LIN {X 0,Y 197.202,Z 363.126,A -85,B 0,C 180,E1 -23005.854,E2 -23005.854} C_VEL
LIN {X 0,Y 193.789,Z 355.62,A -85,B 0,C 180,E1 -23008.882,E2 -23008.882} C_VEL
LIN {X 0,Y 191.136,Z 350.73,A -85,B 0,C 180,E1 -23011.177,E2 -23011.177} C_VEL
LIN {X 0,Y 188.874,Z 346.573,A -85,B 0,C 180,E1 -23013.258,E2 -23013.258} C_VEL
LIN {X 0,Y 185.862,Z 342.068,A -85,B 0,C 180,E1 -23016.015,E2 -23016.015} C_VEL
LIN {X 0,Y 185.125,Z 340.647,A -85,B 0,C 180,E1 -23016.804,E2 -23016.804} C_VEL
LIN {X 0,Y 182.731,Z 338.106,A -85,B 0,C 180,E1 -23019.16,E2 -23019.16} C_VEL
LIN {X 0,Y 181.419,Z 335.441,A -85,B 0,C 180,E1 -23020.775,E2 -23020.775} C_VEL
LIN {X 0,Y 178.641,Z 333.282,A -85,B 0,C 180,E1 -23024.014,E2 -23024.014} C_VEL
LIN {X 0,Y 177.261,Z 330.435,A -85,B 0,C 180,E1 -23026.384,E2 -23026.384} C_VEL
LIN {X 0,Y 177.054,Z 329.764,A -85,B 0,C 180,E1 -23026.806,E2 -23026.806} C_VEL
LIN {X 0,Y 172.985,Z 325.903,A -85,B 0,C 180,E1 -23040,E2 -23040} C_VEL
LIN {X 0,Y 177.156,Z 329.966,A -85,B 0,C 180,E1 -23053.259,E2 -23053.259} C_VEL
LIN {X 0,Y 178.201,Z 332.574,A -85,B 0,C 180,E1 -23055.146,E2 -23055.146} C_VEL
LIN {X 0,Y 181.712,Z 336.354,A -85,B 0,C 180,E1 -23059.486,E2 -23059.486} C_VEL
LIN {X 0,Y 183.271,Z 339.603,A -85,B 0,C 180,E1 -23061.364,E2 -23061.364} C_VEL
LIN {X 0,Y 185.721,Z 342.711,A -85,B 0,C 180,E1 -23063.781,E2 -23063.781} C_VEL
LIN {X 0,Y 187.904,Z 346.733,A -85,B 0,C 180,E1 -23065.921,E2 -23065.921} C_VEL
LIN {X 0,Y 189.084,Z 348.461,A -85,B 0,C 180,E1 -23066.957,E2 -23066.957} C_VEL
LIN {X 0,Y 191.285,Z 352.569,A -85,B 0,C 180,E1 -23068.957,E2 -23068.957} C_VEL
LIN {X 0,Y 194.891,Z 359.939,A -85,B 0,C 180,E1 -23072.134,E2 -23072.134} C_VEL
LIN {X 0,Y 198.257,Z 367.774,A -85,B 0,C 180,E1 -23075.122,E2 -23075.122} C_VEL
LIN {X 0,Y 200.917,Z 375.46,A -85,B 0,C 180,E1 -23077.724,E2 -23077.724} C_VEL
LIN {X 0,Y 202.539,Z 383.023,A -85,B 0,C 180,E1 -23079.938,E2 -23079.938} C_VEL
LIN {X 0,Y 203.603,Z 393.149,A -85,B 0,C 180,E1 -23082.673,E2 -23082.673} C_VEL
LIN {X 0,Y 203.75,Z 403.021,A -85,B 0,C 180,E1 -23085.29,E2 -23085.29} C_VEL
LIN {X 0,Y 203.187,Z 411.249,A -85,B 0,C 180,E1 -23087.478,E2 -23087.478} C_VEL
LIN {X 0,Y 198.333,Z 421.868,A -85,B 0,C 180,E1 -23089.707,E2 -23089.707} C_VEL
LIN {X 0,Y 193.072,Z 432.353,A -85,B 0,C 180,E1 -23092.431,E2 -23092.431} C_VEL
LIN {X 0,Y 187.527,Z 442.605,A -85,B 0,C 180,E1 -23095.794,E2 -23095.794} C_VEL
LIN {X 0,Y 183.46,Z 450.011,A -85,B 0,C 180,E1 -23098.858,E2 -23098.858} C_VEL
LIN {X 0,Y 179.707,Z 456.354,A -85,B 0,C 180,E1 -23102.011,E2 -23102.011} C_VEL
LIN {X 0,Y 175.598,Z 463.314,A -85,B 0,C 180,E1 -23106.407,E2 -23106.407} C_VEL
LIN {X 0,Y 172.589,Z 468.788,A -85,B 0,C 180,E1 -23110.987,E2 -23110.987} C_VEL
LIN {X 0,Y 170.443,Z 472.925,A -85,B 0,C 180,E1 -23115.675,E2 -23115.675} C_VEL
LIN {X 0,Y 169.294,Z 475.826,A -85,B 0,C 180,E1 -23120.441,E2 -23120.441} C_VEL
LIN {X 0,Y 168.85,Z 477.556,A -85,B 0,C 180,E1 -23125.224,E2 -23125.224} C_VEL
LIN {X 0,Y 168.868,Z 478.146,A -85,B 0,C 180,E1 -23129.999,E2 -23129.999} C_VEL
LIN {X 0,Y 168.811,Z 477.96,A -85,B 0,C 180,E1 -23132.539,E2 -23132.539} C_VEL
LIN {X 0,Y 168.123,Z 477.6,A -85,B 0,C 180,E1 -23134.528,E2 -23134.528} C_VEL
LIN {X 0,Y 165.469,Z 476.617,A -85,B 0,C 180,E1 -23137.794,E2 -23137.794} C_VEL
LIN {X 0,Y 163.446,Z 475.488,A -85,B 0,C 180,E1 -23140.46,E2 -23140.46} C_VEL
LIN {X 0,Y 162.86,Z 474.386,A -85,B 0,C 180,E1 -23142.503,E2 -23142.503} C_VEL
LIN {X 0,Y 162.958,Z 473.946,A -85,B 0,C 180,E1 -23143.184,E2 -23143.184} C_VEL
LIN {X 0,Y 165.212,Z 469.819,A -85,B 0,C 180,E1 -23148.604,E2 -23148.604} C_VEL
LIN {X 0,Y 168.096,Z 464.744,A -85,B 0,C 180,E1 -23153.315,E2 -23153.315} C_VEL
LIN {X 0,Y 172.217,Z 458.041,A -85,B 0,C 180,E1 -23157.988,E2 -23157.988} C_VEL
LIN {X 0,Y 176.662,Z 450.925,A -85,B 0,C 180,E1 -23161.809,E2 -23161.809} C_VEL
LIN {X 0,Y 181.724,Z 442.379,A -85,B 0,C 180,E1 -23165.457,E2 -23165.457} C_VEL
LIN {X 0,Y 187.448,Z 432.092,A -85,B 0,C 180,E1 -23168.902,E2 -23168.902} C_VEL
LIN {X 0,Y 192.941,Z 421.569,A -85,B 0,C 180,E1 -23171.662,E2 -23171.662} C_VEL
LIN {X 0,Y 197.1,Z 412.813,A -85,B 0,C 180,E1 -23173.545,E2 -23173.545} C_VEL
LIN {X 0,Y 197.872,Z 405.133,A -85,B 0,C 180,E1 -23175.704,E2 -23175.704} C_VEL
LIN {X 0,Y 197.933,Z 396.156,A -85,B 0,C 180,E1 -23178.212,E2 -23178.212} C_VEL
LIN {X 0,Y 197.384,Z 387.797,A -85,B 0,C 180,E1 -23180.576,E2 -23180.576} C_VEL
LIN {X 0,Y 196.151,Z 380.242,A -85,B 0,C 180,E1 -23182.871,E2 -23182.871} C_VEL
LIN {X 0,Y 193.642,Z 372.121,A -85,B 0,C 180,E1 -23185.768,E2 -23185.768} C_VEL
LIN {X 0,Y 190.07,Z 363.095,A -85,B 0,C 180,E1 -23189.442,E2 -23189.442} C_VEL
LIN {X 0,Y 187.963,Z 358.495,A -85,B 0,C 180,E1 -23191.528,E2 -23191.528} C_VEL
LIN {X 0,Y 185.822,Z 354.199,A -85,B 0,C 180,E1 -23193.722,E2 -23193.722} C_VEL
LIN {X 0,Y 183.236,Z 349.61,A -85,B 0,C 180,E1 -23196.401,E2 -23196.401} C_VEL
LIN {X 0,Y 182.424,Z 348.083,A -85,B 0,C 180,E1 -23197.341,E2 -23197.341} C_VEL
LIN {X 0,Y 180.015,Z 344.398,A -85,B 0,C 180,E1 -23200.08,E2 -23200.08} C_VEL
LIN {X 0,Y 179.298,Z 342.606,A -85,B 0,C 180,E1 -23201.133,E2 -23201.133} C_VEL
LIN {X 0,Y 176.179,Z 338.88,A -85,B 0,C 180,E1 -23205.415,E2 -23205.415} C_VEL
LIN {X 0,Y 175.339,Z 336.621,A -85,B 0,C 180,E1 -23207.117,E2 -23207.117} C_VEL
LIN {X 0,Y 171.676,Z 333.091,A -85,B 0,C 180,E1 -23217.654,E2 -23217.654} C_VEL
LIN {X 0,Y 171.653,Z 332.38,A -85,B 0,C 180,E1 -23220,E2 -23220} C_VEL
LIN {X 0,Y 175.38,Z 336.795,A -85,B 0,C 180,E1 -23233.248,E2 -23233.248} C_VEL
LIN {X 0,Y 176.75,Z 339.926,A -85,B 0,C 180,E1 -23235.865,E2 -23235.865} C_VEL
LIN {X 0,Y 179.396,Z 342.425,A -85,B 0,C 180,E1 -23239.227,E2 -23239.227} C_VEL
LIN {X 0,Y 181.197,Z 345.679,A -85,B 0,C 180,E1 -23241.502,E2 -23241.502} C_VEL
LIN {X 0,Y 182.85,Z 347.535,A -85,B 0,C 180,E1 -23243.215,E2 -23243.215} C_VEL
LIN {X 0,Y 185.131,Z 351.652,A -85,B 0,C 180,E1 -23245.688,E2 -23245.688} C_VEL
LIN {X 0,Y 185.833,Z 352.79,A -85,B 0,C 180,E1 -23246.369,E2 -23246.369} C_VEL
LIN {X 0,Y 188.924,Z 359.018,A -85,B 0,C 180,E1 -23249.532,E2 -23249.532} C_VEL
LIN {X 0,Y 192.163,Z 366.162,A -85,B 0,C 180,E1 -23252.738,E2 -23252.738} C_VEL
LIN {X 0,Y 195.333,Z 374.748,A -85,B 0,C 180,E1 -23256.073,E2 -23256.073} C_VEL
LIN {X 0,Y 197.247,Z 382.066,A -85,B 0,C 180,E1 -23258.574,E2 -23258.574} C_VEL
LIN {X 0,Y 198.42,Z 391.372,A -85,B 0,C 180,E1 -23261.394,E2 -23261.394} C_VEL
LIN {X 0,Y 198.733,Z 400.492,A -85,B 0,C 180,E1 -23264.035,E2 -23264.035} C_VEL
LIN {X 0,Y 198.486,Z 407.964,A -85,B 0,C 180,E1 -23266.215,E2 -23266.215} C_VEL
LIN {X 0,Y 192.617,Z 420.554,A -85,B 0,C 180,E1 -23268.948,E2 -23268.948} C_VEL
LIN {X 0,Y 187.259,Z 430.768,A -85,B 0,C 180,E1 -23271.741,E2 -23271.741} C_VEL
LIN {X 0,Y 181.653,Z 440.752,A -85,B 0,C 180,E1 -23275.205,E2 -23275.205} C_VEL
LIN {X 0,Y 176.564,Z 449.037,A -85,B 0,C 180,E1 -23278.84,E2 -23278.84} C_VEL
LIN {X 0,Y 171.696,Z 456.819,A -85,B 0,C 180,E1 -23283.241,E2 -23283.241} C_VEL
LIN {X 0,Y 167.871,Z 463.012,A -85,B 0,C 180,E1 -23287.866,E2 -23287.866} C_VEL
LIN {X 0,Y 164.968,Z 467.792,A -85,B 0,C 180,E1 -23292.651,E2 -23292.651} C_VEL
LIN {X 0,Y 163.085,Z 471.291,A -85,B 0,C 180,E1 -23297.558,E2 -23297.558} C_VEL
LIN {X 0,Y 162.041,Z 473.601,A -85,B 0,C 180,E1 -23302.525,E2 -23302.525} C_VEL
LIN {X 0,Y 161.762,Z 474.794,A -85,B 0,C 180,E1 -23307.819,E2 -23307.819} C_VEL
LIN {X 0,Y 161.765,Z 474.803,A -85,B 0,C 180,E1 -23312.211,E2 -23312.211} C_VEL
LIN {X 0,Y 162.039,Z 473.656,A -85,B 0,C 180,E1 -23317.477,E2 -23317.477} C_VEL
LIN {X 0,Y 163.07,Z 471.389,A -85,B 0,C 180,E1 -23322.445,E2 -23322.445} C_VEL
LIN {X 0,Y 164.943,Z 467.927,A -85,B 0,C 180,E1 -23327.354,E2 -23327.354} C_VEL
LIN {X 0,Y 167.798,Z 463.189,A -85,B 0,C 180,E1 -23332.146,E2 -23332.146} C_VEL
LIN {X 0,Y 171.647,Z 457.052,A -85,B 0,C 180,E1 -23336.769,E2 -23336.769} C_VEL
LIN {X 0,Y 176.452,Z 449.326,A -85,B 0,C 180,E1 -23341.184,E2 -23341.184} C_VEL
LIN {X 0,Y 181.566,Z 441.089,A -85,B 0,C 180,E1 -23344.816,E2 -23344.816} C_VEL
LIN {X 0,Y 186.262,Z 432.664,A -85,B 0,C 180,E1 -23347.817,E2 -23347.817} C_VEL
LIN {X 0,Y 191.548,Z 422.779,A -85,B 0,C 180,E1 -23350.637,E2 -23350.637} C_VEL
LIN {X 0,Y 197.082,Z 411.356,A -85,B 0,C 180,E1 -23353.242,E2 -23353.242} C_VEL
LIN {X 0,Y 198.443,Z 408.394,A -85,B 0,C 180,E1 -23353.839,E2 -23353.839} C_VEL
LIN {X 0,Y 198.877,Z 399.443,A -85,B 0,C 180,E1 -23356.401,E2 -23356.401} C_VEL
LIN {X 0,Y 198.352,Z 389.337,A -85,B 0,C 180,E1 -23359.376,E2 -23359.376} C_VEL
LIN {X 0,Y 197.048,Z 380.688,A -85,B 0,C 180,E1 -23362.03,E2 -23362.03} C_VEL
LIN {X 0,Y 195.163,Z 374.105,A -85,B 0,C 180,E1 -23364.353,E2 -23364.353} C_VEL
LIN {X 0,Y 191.786,Z 365.097,A -85,B 0,C 180,E1 -23367.902,E2 -23367.902} C_VEL
LIN {X 0,Y 188.648,Z 358.233,A -85,B 0,C 180,E1 -23371.033,E2 -23371.033} C_VEL
LIN {X 0,Y 185.32,Z 351.886,A -85,B 0,C 180,E1 -23374.418,E2 -23374.418} C_VEL
LIN {X 0,Y 182.981,Z 347.82,A -85,B 0,C 180,E1 -23376.928,E2 -23376.928} C_VEL
LIN {X 0,Y 182.386,Z 346.853,A -85,B 0,C 180,E1 -23377.604,E2 -23377.604} C_VEL
LIN {X 0,Y 180.165,Z 344.134,A -85,B 0,C 180,E1 -23380.042,E2 -23380.042} C_VEL
LIN {X 0,Y 179.184,Z 342.058,A -85,B 0,C 180,E1 -23381.427,E2 -23381.427} C_VEL
LIN {X 0,Y 176.663,Z 339.791,A -85,B 0,C 180,E1 -23384.719,E2 -23384.719} C_VEL
LIN {X 0,Y 175.323,Z 336.612,A -85,B 0,C 180,E1 -23387.41,E2 -23387.41} C_VEL
LIN {X 0,Y 171.879,Z 332.904,A -85,B 0,C 180,E1 -23400,E2 -23400} C_VEL
LIN {X 0,Y 175.446,Z 336.802,A -85,B 0,C 180,E1 -23412.654,E2 -23412.654} C_VEL
LIN {X 0,Y 176.898,Z 340.033,A -85,B 0,C 180,E1 -23415.408,E2 -23415.408} C_VEL
LIN {X 0,Y 179.479,Z 342.97,A -85,B 0,C 180,E1 -23418.847,E2 -23418.847} C_VEL
LIN {X 0,Y 181.297,Z 346.656,A -85,B 0,C 180,E1 -23421.236,E2 -23421.236} C_VEL
LIN {X 0,Y 182.985,Z 348.837,A -85,B 0,C 180,E1 -23423.034,E2 -23423.034} C_VEL
LIN {X 0,Y 185.01,Z 352.876,A -85,B 0,C 180,E1 -23425.31,E2 -23425.31} C_VEL
LIN {X 0,Y 185.932,Z 354.337,A -85,B 0,C 180,E1 -23426.195,E2 -23426.195} C_VEL
LIN {X 0,Y 188.606,Z 359.937,A -85,B 0,C 180,E1 -23428.974,E2 -23428.974} C_VEL
LIN {X 0,Y 191.739,Z 367.012,A -85,B 0,C 180,E1 -23432.107,E2 -23432.107} C_VEL
LIN {X 0,Y 195.069,Z 376.14,A -85,B 0,C 180,E1 -23435.615,E2 -23435.615} C_VEL
LIN {X 0,Y 196.873,Z 383.3,A -85,B 0,C 180,E1 -23438.009,E2 -23438.009} C_VEL
LIN {X 0,Y 197.883,Z 391.888,A -85,B 0,C 180,E1 -23440.523,E2 -23440.523} C_VEL
LIN {X 0,Y 198.12,Z 402.137,A -85,B 0,C 180,E1 -23443.425,E2 -23443.425} C_VEL
LIN {X 0,Y 197.495,Z 411.403,A -85,B 0,C 180,E1 -23446.017,E2 -23446.017} C_VEL
LIN {X 0,Y 197.18,Z 412.94,A -85,B 0,C 180,E1 -23446.435,E2 -23446.435} C_VEL
LIN {X 0,Y 192.002,Z 423.699,A -85,B 0,C 180,E1 -23448.786,E2 -23448.786} C_VEL
LIN {X 0,Y 186.581,Z 433.914,A -85,B 0,C 180,E1 -23451.573,E2 -23451.573} C_VEL
LIN {X 0,Y 180.919,Z 443.892,A -85,B 0,C 180,E1 -23455.041,E2 -23455.041} C_VEL
LIN {X 0,Y 175.943,Z 452.18,A -85,B 0,C 180,E1 -23458.715,E2 -23458.715} C_VEL
LIN {X 0,Y 171.103,Z 459.964,A -85,B 0,C 180,E1 -23463.139,E2 -23463.139} C_VEL
LIN {X 0,Y 167.283,Z 466.157,A -85,B 0,C 180,E1 -23467.782,E2 -23467.782} C_VEL
LIN {X 0,Y 164.601,Z 470.948,A -85,B 0,C 180,E1 -23472.609,E2 -23472.609} C_VEL
LIN {X 0,Y 162.775,Z 474.457,A -85,B 0,C 180,E1 -23477.532,E2 -23477.532} C_VEL
LIN {X 0,Y 161.907,Z 476.765,A -85,B 0,C 180,E1 -23482.517,E2 -23482.517} C_VEL
LIN {X 0,Y 161.712,Z 477.925,A -85,B 0,C 180,E1 -23487.508,E2 -23487.508} C_VEL
LIN {X 0,Y 161.772,Z 478.077,A -85,B 0,C 180,E1 -23489.999,E2 -23489.999} C_VEL
LIN {X 0,Y 161.749,Z 477.471,A -85,B 0,C 180,E1 -23494.984,E2 -23494.984} C_VEL
LIN {X 0,Y 162.246,Z 475.72,A -85,B 0,C 180,E1 -23499.977,E2 -23499.977} C_VEL
LIN {X 0,Y 162.958,Z 473.946,A -85,B 0,C 180,E1 -23503.184,E2 -23503.184} C_VEL
LIN {X 0,Y 162.928,Z 472.66,A -85,B 0,C 180,E1 -23505.21,E2 -23505.21} C_VEL
LIN {X 0,Y 161.471,Z 470.171,A -85,B 0,C 180,E1 -23508.572,E2 -23508.572} C_VEL
LIN {X 0,Y 160.53,Z 467.889,A -85,B 0,C 180,E1 -23511.268,E2 -23511.268} C_VEL
LIN {X 0,Y 160.819,Z 465.914,A -85,B 0,C 180,E1 -23513.257,E2 -23513.257} C_VEL
LIN {X 0,Y 161.214,Z 465.172,A -85,B 0,C 180,E1 -23513.895,E2 -23513.895} C_VEL
LIN {X 0,Y 164.741,Z 459.785,A -85,B 0,C 180,E1 -23517.985,E2 -23517.985} C_VEL
LIN {X 0,Y 169.886,Z 451.972,A -85,B 0,C 180,E1 -23522.532,E2 -23522.532} C_VEL
LIN {X 0,Y 175.142,Z 443.663,A -85,B 0,C 180,E1 -23526.289,E2 -23526.289} C_VEL
LIN {X 0,Y 181.039,Z 433.65,A -85,B 0,C 180,E1 -23529.83,E2 -23529.83} C_VEL
LIN {X 0,Y 186.679,Z 423.415,A -85,B 0,C 180,E1 -23532.659,E2 -23532.659} C_VEL
LIN {X 0,Y 191.32,Z 414.102,A -85,B 0,C 180,E1 -23534.739,E2 -23534.739} C_VEL
LIN {X 0,Y 192.255,Z 405.43,A -85,B 0,C 180,E1 -23537.322,E2 -23537.322} C_VEL
LIN {X 0,Y 192.424,Z 396.069,A -85,B 0,C 180,E1 -23540.082,E2 -23540.082} C_VEL
LIN {X 0,Y 191.739,Z 387.291,A -85,B 0,C 180,E1 -23542.786,E2 -23542.786} C_VEL
LIN {X 0,Y 190.786,Z 382.413,A -85,B 0,C 180,E1 -23544.471,E2 -23544.471} C_VEL
LIN {X 0,Y 188.145,Z 373.913,A -85,B 0,C 180,E1 -23547.831,E2 -23547.831} C_VEL
LIN {X 0,Y 185.351,Z 366.665,A -85,B 0,C 180,E1 -23551.09,E2 -23551.09} C_VEL
LIN {X 0,Y 183.951,Z 363.455,A -85,B 0,C 180,E1 -23552.712,E2 -23552.712} C_VEL
LIN {X 0,Y 182.129,Z 359.312,A -85,B 0,C 180,E1 -23554.883,E2 -23554.883} C_VEL
LIN {X 0,Y 179.023,Z 353.491,A -85,B 0,C 180,E1 -23558.677,E2 -23558.677} C_VEL
LIN {X 0,Y 177.081,Z 349.657,A -85,B 0,C 180,E1 -23561.413,E2 -23561.413} C_VEL
LIN {X 0,Y 176.507,Z 348.722,A -85,B 0,C 180,E1 -23562.251,E2 -23562.251} C_VEL
LIN {X 0,Y 174.052,Z 345.296,A -85,B 0,C 180,E1 -23566.129,E2 -23566.129} C_VEL
LIN {X 0,Y 173.385,Z 343.412,A -85,B 0,C 180,E1 -23567.714,E2 -23567.714} C_VEL
LIN {X 0,Y 170.284,Z 339.364,A -85,B 0,C 180,E1 -23580,E2 -23580} C_VEL
LIN {X 0,Y 173.479,Z 343.686,A -85,B 0,C 180,E1 -23592.838,E2 -23592.838} C_VEL
LIN {X 0,Y 174.663,Z 346.541,A -85,B 0,C 180,E1 -23595.371,E2 -23595.371} C_VEL
LIN {X 0,Y 177.038,Z 349.075,A -85,B 0,C 180,E1 -23598.742,E2 -23598.742} C_VEL
LIN {X 0,Y 178.89,Z 352.406,A -85,B 0,C 180,E1 -23601.305,E2 -23601.305} C_VEL
LIN {X 0,Y 180.281,Z 354.423,A -85,B 0,C 180,E1 -23602.945,E2 -23602.945} C_VEL
LIN {X 0,Y 182.992,Z 359.756,A -85,B 0,C 180,E1 -23606.211,E2 -23606.211} C_VEL
LIN {X 0,Y 186.024,Z 366.289,A -85,B 0,C 180,E1 -23609.668,E2 -23609.668} C_VEL
LIN {X 0,Y 189.15,Z 374.497,A -85,B 0,C 180,E1 -23613.327,E2 -23613.327} C_VEL
LIN {X 0,Y 191.543,Z 382.722,A -85,B 0,C 180,E1 -23616.535,E2 -23616.535} C_VEL
LIN {X 0,Y 192.65,Z 389.546,A -85,B 0,C 180,E1 -23618.847,E2 -23618.847} C_VEL
LIN {X 0,Y 193.116,Z 398.307,A -85,B 0,C 180,E1 -23621.593,E2 -23621.593} C_VEL
LIN {X 0,Y 192.782,Z 408.307,A -85,B 0,C 180,E1 -23624.652,E2 -23624.652} C_VEL
LIN {X 0,Y 192.583,Z 409.836,A -85,B 0,C 180,E1 -23625.12,E2 -23625.12} C_VEL
LIN {X 0,Y 187.283,Z 420.627,A -85,B 0,C 180,E1 -23627.511,E2 -23627.511} C_VEL
LIN {X 0,Y 181.691,Z 430.837,A -85,B 0,C 180,E1 -23630.342,E2 -23630.342} C_VEL
LIN {X 0,Y 175.847,Z 440.823,A -85,B 0,C 180,E1 -23633.88,E2 -23633.88} C_VEL
LIN {X 0,Y 170.465,Z 449.109,A -85,B 0,C 180,E1 -23637.592,E2 -23637.592} C_VEL
LIN {X 0,Y 165.341,Z 456.89,A -85,B 0,C 180,E1 -23642.125,E2 -23642.125} C_VEL
LIN {X 0,Y 161.275,Z 463.083,A -85,B 0,C 180,E1 -23646.91,E2 -23646.91} C_VEL
LIN {X 0,Y 158.184,Z 467.863,A -85,B 0,C 180,E1 -23651.882,E2 -23651.882} C_VEL
LIN {X 0,Y 156.126,Z 471.361,A -85,B 0,C 180,E1 -23656.994,E2 -23656.994} C_VEL
LIN {X 0,Y 154.985,Z 473.671,A -85,B 0,C 180,E1 -23662.182,E2 -23662.182} C_VEL
LIN {X 0,Y 154.667,Z 474.844,A -85,B 0,C 180,E1 -23667.397,E2 -23667.397} C_VEL
LIN {X 0,Y 154.657,Z 474.933,A -85,B 0,C 180,E1 -23671.302,E2 -23671.302} C_VEL
LIN {X 0,Y 154.758,Z 474.43,A -85,B 0,C 180,E1 -23675.212,E2 -23675.212} C_VEL
LIN {X 0,Y 155.451,Z 472.737,A -85,B 0,C 180,E1 -23680.42,E2 -23680.42} C_VEL
LIN {X 0,Y 156.953,Z 469.881,A -85,B 0,C 180,E1 -23685.586,E2 -23685.586} C_VEL
LIN {X 0,Y 159.571,Z 465.792,A -85,B 0,C 180,E1 -23690.632,E2 -23690.632} C_VEL
LIN {X 0,Y 163.115,Z 460.374,A -85,B 0,C 180,E1 -23695.523,E2 -23695.523} C_VEL
LIN {X 0,Y 167.723,Z 453.47,A -85,B 0,C 180,E1 -23700.188,E2 -23700.188} C_VEL
LIN {X 0,Y 172.594,Z 446.052,A -85,B 0,C 180,E1 -23704.049,E2 -23704.049} C_VEL
LIN {X 0,Y 177.38,Z 438.369,A -85,B 0,C 180,E1 -23707.221,E2 -23707.221} C_VEL
LIN {X 0,Y 183.381,Z 427.991,A -85,B 0,C 180,E1 -23710.656,E2 -23710.656} C_VEL
LIN {X 0,Y 189.09,Z 417.236,A -85,B 0,C 180,E1 -23713.441,E2 -23713.441} C_VEL
LIN {X 0,Y 192.503,Z 410.272,A -85,B 0,C 180,E1 -23714.934,E2 -23714.934} C_VEL
LIN {X 0,Y 193.171,Z 403.449,A -85,B 0,C 180,E1 -23716.984,E2 -23716.984} C_VEL
LIN {X 0,Y 193.078,Z 394.18,A -85,B 0,C 180,E1 -23719.854,E2 -23719.854} C_VEL
LIN {X 0,Y 192.36,Z 386.633,A -85,B 0,C 180,E1 -23722.268,E2 -23722.268} C_VEL
LIN {X 0,Y 190.973,Z 380.214,A -85,B 0,C 180,E1 -23724.576,E2 -23724.576} C_VEL
LIN {X 0,Y 188.448,Z 372.438,A -85,B 0,C 180,E1 -23727.754,E2 -23727.754} C_VEL
LIN {X 0,Y 185.558,Z 365.156,A -85,B 0,C 180,E1 -23731.124,E2 -23731.124} C_VEL
LIN {X 0,Y 182.324,Z 358.13,A -85,B 0,C 180,E1 -23734.911,E2 -23734.911} C_VEL
LIN {X 0,Y 180.174,Z 354.158,A -85,B 0,C 180,E1 -23737.524,E2 -23737.524} C_VEL
LIN {X 0,Y 177.282,Z 349.676,A -85,B 0,C 180,E1 -23741.221,E2 -23741.221} C_VEL
LIN {X 0,Y 176.765,Z 348.59,A -85,B 0,C 180,E1 -23742.053,E2 -23742.053} C_VEL
LIN {X 0,Y 174.463,Z 346.146,A -85,B 0,C 180,E1 -23745.478,E2 -23745.478} C_VEL
LIN {X 0,Y 173.356,Z 343.391,A -85,B 0,C 180,E1 -23748.008,E2 -23748.008} C_VEL
LIN {X 0,Y 170.485,Z 339.883,A -85,B 0,C 180,E1 -23760,E2 -23760} C_VEL
LIN {X 0,Y 173.545,Z 343.561,A -85,B 0,C 180,E1 -23772.127,E2 -23772.127} C_VEL
LIN {X 0,Y 174.962,Z 346.869,A -85,B 0,C 180,E1 -23775.136,E2 -23775.136} C_VEL
LIN {X 0,Y 177.027,Z 349.293,A -85,B 0,C 180,E1 -23778.143,E2 -23778.143} C_VEL
LIN {X 0,Y 178.611,Z 352.906,A -85,B 0,C 180,E1 -23780.589,E2 -23780.589} C_VEL
LIN {X 0,Y 180.233,Z 355.367,A -85,B 0,C 180,E1 -23782.528,E2 -23782.528} C_VEL
LIN {X 0,Y 182.748,Z 360.544,A -85,B 0,C 180,E1 -23785.635,E2 -23785.635} C_VEL
LIN {X 0,Y 185.041,Z 365.749,A -85,B 0,C 180,E1 -23788.343,E2 -23788.343} C_VEL
LIN {X 0,Y 187.832,Z 372.798,A -85,B 0,C 180,E1 -23791.589,E2 -23791.589} C_VEL
LIN {X 0,Y 190.464,Z 380.94,A -85,B 0,C 180,E1 -23794.885,E2 -23794.885} C_VEL
LIN {X 0,Y 191.855,Z 387.457,A -85,B 0,C 180,E1 -23797.186,E2 -23797.186} C_VEL
LIN {X 0,Y 192.468,Z 394.574,A -85,B 0,C 180,E1 -23799.399,E2 -23799.399} C_VEL
LIN {X 0,Y 192.462,Z 404.518,A -85,B 0,C 180,E1 -23802.356,E2 -23802.356} C_VEL
LIN {X 0,Y 191.581,Z 413.544,A -85,B 0,C 180,E1 -23805.054,E2 -23805.054} C_VEL
LIN {X 0,Y 186.695,Z 423.633,A -85,B 0,C 180,E1 -23807.344,E2 -23807.344} C_VEL
LIN {X 0,Y 181.038,Z 433.847,A -85,B 0,C 180,E1 -23810.168,E2 -23810.168} C_VEL
LIN {X 0,Y 175.068,Z 443.825,A -85,B 0,C 180,E1 -23813.691,E2 -23813.691} C_VEL
LIN {X 0,Y 170.645,Z 450.994,A -85,B 0,C 180,E1 -23816.927,E2 -23816.927} C_VEL
LIN {X 0,Y 165.948,Z 458.083,A -85,B 0,C 180,E1 -23820.854,E2 -23820.854} C_VEL
LIN {X 0,Y 161.588,Z 464.662,A -85,B 0,C 180,E1 -23825.596,E2 -23825.596} C_VEL
LIN {X 0,Y 158.443,Z 469.808,A -85,B 0,C 180,E1 -23830.568,E2 -23830.568} C_VEL
LIN {X 0,Y 156.615,Z 472.787,A -85,B 0,C 180,E1 -23834.38,E2 -23834.38} C_VEL
LIN {X 0,Y 155.221,Z 475.688,A -85,B 0,C 180,E1 -23839.565,E2 -23839.565} C_VEL
LIN {X 0,Y 154.679,Z 477.418,A -85,B 0,C 180,E1 -23844.785,E2 -23844.785} C_VEL
LIN {X 0,Y 154.684,Z 478.009,A -85,B 0,C 180,E1 -23849.999,E2 -23849.999} C_VEL
LIN {X 0,Y 154.679,Z 477.401,A -85,B 0,C 180,E1 -23855.213,E2 -23855.213} C_VEL
LIN {X 0,Y 155.22,Z 475.65,A -85,B 0,C 180,E1 -23860.433,E2 -23860.433} C_VEL
LIN {X 0,Y 156.614,Z 472.733,A -85,B 0,C 180,E1 -23865.618,E2 -23865.618} C_VEL
LIN {X 0,Y 159.12,Z 468.581,A -85,B 0,C 180,E1 -23870.691,E2 -23870.691} C_VEL
LIN {X 0,Y 161.214,Z 465.172,A -85,B 0,C 180,E1 -23873.895,E2 -23873.895} C_VEL
LIN {X 0,Y 162.07,Z 462.963,A -85,B 0,C 180,E1 -23875.815,E2 -23875.815} C_VEL
LIN {X 0,Y 162.041,Z 459.127,A -85,B 0,C 180,E1 -23879.059,E2 -23879.059} C_VEL
LIN {X 0,Y 162.47,Z 454.814,A -85,B 0,C 180,E1 -23882.207,E2 -23882.207} C_VEL
LIN {X 0,Y 163.983,Z 451.822,A -85,B 0,C 180,E1 -23883.91,E2 -23883.91} C_VEL
LIN {X 0,Y 169.413,Z 443.591,A -85,B 0,C 180,E1 -23887.725,E2 -23887.725} C_VEL
LIN {X 0,Y 175.609,Z 433.578,A -85,B 0,C 180,E1 -23891.324,E2 -23891.324} C_VEL
LIN {X 0,Y 181.499,Z 423.343,A -85,B 0,C 180,E1 -23894.184,E2 -23894.184} C_VEL
LIN {X 0,Y 185.63,Z 415.418,A -85,B 0,C 180,E1 -23895.998,E2 -23895.998} C_VEL
LIN {X 0,Y 186.816,Z 405.122,A -85,B 0,C 180,E1 -23899.242,E2 -23899.242} C_VEL
LIN {X 0,Y 186.961,Z 395.979,A -85,B 0,C 180,E1 -23902.127,E2 -23902.127} C_VEL
LIN {X 0,Y 186.288,Z 388.491,A -85,B 0,C 180,E1 -23904.672,E2 -23904.672} C_VEL
LIN {X 0,Y 184.412,Z 380.867,A -85,B 0,C 180,E1 -23907.755,E2 -23907.755} C_VEL
LIN {X 0,Y 182.01,Z 373.459,A -85,B 0,C 180,E1 -23911.141,E2 -23911.141} C_VEL
LIN {X 0,Y 180.265,Z 368.992,A -85,B 0,C 180,E1 -23913.487,E2 -23913.487} C_VEL
LIN {X 0,Y 178.734,Z 365.116,A -85,B 0,C 180,E1 -23915.615,E2 -23915.615} C_VEL
LIN {X 0,Y 176.34,Z 360.052,A -85,B 0,C 180,E1 -23918.98,E2 -23918.98} C_VEL
LIN {X 0,Y 174.825,Z 357.22,A -85,B 0,C 180,E1 -23921.24,E2 -23921.24} C_VEL
LIN {X 0,Y 174.277,Z 355.473,A -85,B 0,C 180,E1 -23922.395,E2 -23922.395} C_VEL
LIN {X 0,Y 171.821,Z 351.852,A -85,B 0,C 180,E1 -23926.623,E2 -23926.623} C_VEL
LIN {X 0,Y 171.28,Z 350.145,A -85,B 0,C 180,E1 -23928.161,E2 -23928.161} C_VEL
LIN {X 0,Y 168.618,Z 346.306,A -85,B 0,C 180,E1 -23940,E2 -23940} C_VEL
LIN {X 0,Y 171.304,Z 350.406,A -85,B 0,C 180,E1 -23952.363,E2 -23952.363} C_VEL
LIN {X 0,Y 171.985,Z 352.416,A -85,B 0,C 180,E1 -23954.193,E2 -23954.193} C_VEL
LIN {X 0,Y 174.069,Z 354.973,A -85,B 0,C 180,E1 -23957.627,E2 -23957.627} C_VEL
LIN {X 0,Y 177.107,Z 360.311,A -85,B 0,C 180,E1 -23962.147,E2 -23962.147} C_VEL
LIN {X 0,Y 179.507,Z 365.504,A -85,B 0,C 180,E1 -23965.51,E2 -23965.51} C_VEL
LIN {X 0,Y 182.021,Z 371.568,A -85,B 0,C 180,E1 -23968.858,E2 -23968.858} C_VEL
LIN {X 0,Y 184.46,Z 378.686,A -85,B 0,C 180,E1 -23972.236,E2 -23972.236} C_VEL
LIN {X 0,Y 186.639,Z 387.168,A -85,B 0,C 180,E1 -23975.754,E2 -23975.754} C_VEL
LIN {X 0,Y 187.418,Z 393.593,A -85,B 0,C 180,E1 -23978.052,E2 -23978.052} C_VEL
LIN {X 0,Y 187.566,Z 402.192,A -85,B 0,C 180,E1 -23980.88,E2 -23980.88} C_VEL
LIN {X 0,Y 186.971,Z 410.588,A -85,B 0,C 180,E1 -23983.628,E2 -23983.628} C_VEL
LIN {X 0,Y 186.182,Z 412.779,A -85,B 0,C 180,E1 -23984.177,E2 -23984.177} C_VEL
LIN {X 0,Y 180.092,Z 424.257,A -85,B 0,C 180,E1 -23986.929,E2 -23986.929} C_VEL
LIN {X 0,Y 173.942,Z 434.74,A -85,B 0,C 180,E1 -23990.146,E2 -23990.146} C_VEL
LIN {X 0,Y 168.482,Z 443.387,A -85,B 0,C 180,E1 -23993.531,E2 -23993.531} C_VEL
LIN {X 0,Y 163.043,Z 451.274,A -85,B 0,C 180,E1 -23997.399,E2 -23997.399} C_VEL
LIN {X 0,Y 157.867,Z 458.636,A -85,B 0,C 180,E1 -24002.133,E2 -24002.133} C_VEL
LIN {X 0,Y 153.778,Z 464.475,A -85,B 0,C 180,E1 -24007.142,E2 -24007.142} C_VEL
LIN {X 0,Y 151.429,Z 467.933,A -85,B 0,C 180,E1 -24011.043,E2 -24011.043} C_VEL
LIN {X 0,Y 149.166,Z 471.431,A -85,B 0,C 180,E1 -24016.376,E2 -24016.376} C_VEL
LIN {X 0,Y 147.952,Z 473.74,A -85,B 0,C 180,E1 -24021.808,E2 -24021.808} C_VEL
LIN {X 0,Y 147.571,Z 474.913,A -85,B 0,C 180,E1 -24027.271,E2 -24027.271} C_VEL
LIN {X 0,Y 147.597,Z 475.045,A -85,B 0,C 180,E1 -24030.614,E2 -24030.614} C_VEL
LIN {X 0,Y 147.69,Z 474.499,A -85,B 0,C 180,E1 -24035.462,E2 -24035.462} C_VEL
LIN {X 0,Y 148.459,Z 472.805,A -85,B 0,C 180,E1 -24040.916,E2 -24040.916} C_VEL
LIN {X 0,Y 150.081,Z 469.95,A -85,B 0,C 180,E1 -24046.319,E2 -24046.319} C_VEL
LIN {X 0,Y 152.876,Z 465.861,A -85,B 0,C 180,E1 -24051.579,E2 -24051.579} C_VEL
LIN {X 0,Y 156.678,Z 460.442,A -85,B 0,C 180,E1 -24056.652,E2 -24056.652} C_VEL
LIN {X 0,Y 161.585,Z 453.538,A -85,B 0,C 180,E1 -24061.462,E2 -24061.462} C_VEL
LIN {X 0,Y 166.746,Z 446.119,A -85,B 0,C 180,E1 -24065.418,E2 -24065.418} C_VEL
LIN {X 0,Y 172.258,Z 437.536,A -85,B 0,C 180,E1 -24069.027,E2 -24069.027} C_VEL
LIN {X 0,Y 178.03,Z 428.058,A -85,B 0,C 180,E1 -24072.152,E2 -24072.152} C_VEL
LIN {X 0,Y 183.975,Z 417.302,A -85,B 0,C 180,E1 -24074.969,E2 -24074.969} C_VEL
LIN {X 0,Y 186.625,Z 412.15,A -85,B 0,C 180,E1 -24076.1,E2 -24076.1} C_VEL
LIN {X 0,Y 187.124,Z 410.108,A -85,B 0,C 180,E1 -24076.689,E2 -24076.689} C_VEL
LIN {X 0,Y 187.691,Z 401.129,A -85,B 0,C 180,E1 -24079.618,E2 -24079.618} C_VEL
LIN {X 0,Y 187.431,Z 392.602,A -85,B 0,C 180,E1 -24082.46,E2 -24082.46} C_VEL
LIN {X 0,Y 186.787,Z 387.435,A -85,B 0,C 180,E1 -24084.324,E2 -24084.324} C_VEL
LIN {X 0,Y 185.146,Z 380.615,A -85,B 0,C 180,E1 -24087.109,E2 -24087.109} C_VEL
LIN {X 0,Y 182.652,Z 373.035,A -85,B 0,C 180,E1 -24090.62,E2 -24090.62} C_VEL
LIN {X 0,Y 180.406,Z 367.408,A -85,B 0,C 180,E1 -24093.637,E2 -24093.637} C_VEL
LIN {X 0,Y 178.936,Z 363.949,A -85,B 0,C 180,E1 -24095.644,E2 -24095.644} C_VEL
LIN {X 0,Y 176.494,Z 359.295,A -85,B 0,C 180,E1 -24098.999,E2 -24098.999} C_VEL
LIN {X 0,Y 174.919,Z 356.788,A -85,B 0,C 180,E1 -24101.25,E2 -24101.25} C_VEL
LIN {X 0,Y 174.341,Z 355.205,A -85,B 0,C 180,E1 -24102.402,E2 -24102.402} C_VEL
LIN {X 0,Y 171.833,Z 351.976,A -85,B 0,C 180,E1 -24106.699,E2 -24106.699} C_VEL
LIN {X 0,Y 171.236,Z 350.112,A -85,B 0,C 180,E1 -24108.458,E2 -24108.458} C_VEL
LIN {X 0,Y 168.808,Z 346.804,A -85,B 0,C 180,E1 -24120,E2 -24120} C_VEL
LIN {X 0,Y 171.435,Z 350.289,A -85,B 0,C 180,E1 -24131.674,E2 -24131.674} C_VEL
LIN {X 0,Y 172.37,Z 352.976,A -85,B 0,C 180,E1 -24134.16,E2 -24134.16} C_VEL
LIN {X 0,Y 174.435,Z 355.814,A -85,B 0,C 180,E1 -24137.588,E2 -24137.588} C_VEL
LIN {X 0,Y 175.7,Z 358.976,A -85,B 0,C 180,E1 -24139.877,E2 -24139.877} C_VEL
LIN {X 0,Y 177.308,Z 361.922,A -85,B 0,C 180,E1 -24142.12,E2 -24142.12} C_VEL
LIN {X 0,Y 179.288,Z 366.324,A -85,B 0,C 180,E1 -24144.922,E2 -24144.922} C_VEL
LIN {X 0,Y 181.324,Z 371.502,A -85,B 0,C 180,E1 -24147.717,E2 -24147.717} C_VEL
LIN {X 0,Y 183.766,Z 378.519,A -85,B 0,C 180,E1 -24151.084,E2 -24151.084} C_VEL
LIN {X 0,Y 186.01,Z 386.631,A -85,B 0,C 180,E1 -24154.523,E2 -24154.523} C_VEL
LIN {X 0,Y 186.86,Z 392.34,A -85,B 0,C 180,E1 -24156.585,E2 -24156.585} C_VEL
LIN {X 0,Y 187.08,Z 400.516,A -85,B 0,C 180,E1 -24159.245,E2 -24159.245} C_VEL
LIN {X 0,Y 186.58,Z 409.262,A -85,B 0,C 180,E1 -24162.001,E2 -24162.001} C_VEL
LIN {X 0,Y 185.658,Z 415.683,A -85,B 0,C 180,E1 -24164.008,E2 -24164.008} C_VEL
LIN {X 0,Y 179.496,Z 427.136,A -85,B 0,C 180,E1 -24166.749,E2 -24166.749} C_VEL
LIN {X 0,Y 173.756,Z 436.774,A -85,B 0,C 180,E1 -24169.672,E2 -24169.672} C_VEL
LIN {X 0,Y 168.441,Z 445.188,A -85,B 0,C 180,E1 -24172.88,E2 -24172.88} C_VEL
LIN {X 0,Y 163.927,Z 452.045,A -85,B 0,C 180,E1 -24176.127,E2 -24176.127} C_VEL
LIN {X 0,Y 158.464,Z 459.828,A -85,B 0,C 180,E1 -24180.799,E2 -24180.799} C_VEL
LIN {X 0,Y 154.044,Z 466.111,A -85,B 0,C 180,E1 -24185.847,E2 -24185.847} C_VEL
LIN {X 0,Y 151.013,Z 470.81,A -85,B 0,C 180,E1 -24190.987,E2 -24190.987} C_VEL
LIN {X 0,Y 148.847,Z 474.319,A -85,B 0,C 180,E1 -24196.344,E2 -24196.344} C_VEL
LIN {X 0,Y 147.786,Z 476.627,A -85,B 0,C 180,E1 -24201.797,E2 -24201.797} C_VEL
LIN {X 0,Y 147.525,Z 477.787,A -85,B 0,C 180,E1 -24207.268,E2 -24207.268} C_VEL
LIN {X 0,Y 147.587,Z 477.94,A -85,B 0,C 180,E1 -24209.999,E2 -24209.999} C_VEL
LIN {X 0,Y 147.606,Z 477.332,A -85,B 0,C 180,E1 -24215.463,E2 -24215.463} C_VEL
LIN {X 0,Y 148.216,Z 475.581,A -85,B 0,C 180,E1 -24220.932,E2 -24220.932} C_VEL
LIN {X 0,Y 149.737,Z 472.662,A -85,B 0,C 180,E1 -24226.355,E2 -24226.355} C_VEL
LIN {X 0,Y 152.446,Z 468.511,A -85,B 0,C 180,E1 -24231.641,E2 -24231.641} C_VEL
LIN {X 0,Y 156.167,Z 463.012,A -85,B 0,C 180,E1 -24236.744,E2 -24236.744} C_VEL
LIN {X 0,Y 161.048,Z 456.02,A -85,B 0,C 180,E1 -24241.577,E2 -24241.577} C_VEL
LIN {X 0,Y 163.983,Z 451.822,A -85,B 0,C 180,E1 -24243.91,E2 -24243.91} C_VEL
LIN {X 0,Y 164.824,Z 449.788,A -85,B 0,C 180,E1 -24245.062,E2 -24245.062} C_VEL
LIN {X 0,Y 164.539,Z 446.605,A -85,B 0,C 180,E1 -24247.146,E2 -24247.146} C_VEL
LIN {X 0,Y 164.421,Z 443.323,A -85,B 0,C 180,E1 -24249.202,E2 -24249.202} C_VEL
LIN {X 0,Y 165.48,Z 440.973,A -85,B 0,C 180,E1 -24250.267,E2 -24250.267} C_VEL
LIN {X 0,Y 171.309,Z 431.876,A -85,B 0,C 180,E1 -24253.405,E2 -24253.405} C_VEL
LIN {X 0,Y 177.537,Z 421.352,A -85,B 0,C 180,E1 -24256.254,E2 -24256.254} C_VEL
LIN {X 0,Y 180.045,Z 416.413,A -85,B 0,C 180,E1 -24257.456,E2 -24257.456} C_VEL
LIN {X 0,Y 181.252,Z 407.355,A -85,B 0,C 180,E1 -24260.464,E2 -24260.464} C_VEL
LIN {X 0,Y 181.674,Z 399.326,A -85,B 0,C 180,E1 -24263.16,E2 -24263.16} C_VEL
LIN {X 0,Y 181.264,Z 392.122,A -85,B 0,C 180,E1 -24265.776,E2 -24265.776} C_VEL
LIN {X 0,Y 179.421,Z 383.912,A -85,B 0,C 180,E1 -24269.389,E2 -24269.389} C_VEL
LIN {X 0,Y 176.951,Z 375.65,A -85,B 0,C 180,E1 -24273.525,E2 -24273.525} C_VEL
LIN {X 0,Y 175.2,Z 370.829,A -85,B 0,C 180,E1 -24276.351,E2 -24276.351} C_VEL
LIN {X 0,Y 173.063,Z 365.897,A -85,B 0,C 180,E1 -24279.807,E2 -24279.807} C_VEL
LIN {X 0,Y 171.27,Z 361.536,A -85,B 0,C 180,E1 -24283.307,E2 -24283.307} C_VEL
LIN {X 0,Y 169.454,Z 358.658,A -85,B 0,C 180,E1 -24286.814,E2 -24286.814} C_VEL
LIN {X 0,Y 169.09,Z 357.402,A -85,B 0,C 180,E1 -24288.006,E2 -24288.006} C_VEL
LIN {X 0,Y 168.131,Z 356.244,A -85,B 0,C 180,E1 -24290.375,E2 -24290.375} C_VEL
LIN {X 0,Y 166.657,Z 353.154,A -85,B 0,C 180,E1 -24300,E2 -24300} C_VEL
LIN {X 0,Y 168.933,Z 357.112,A -85,B 0,C 180,E1 -24312.006,E2 -24312.006} C_VEL
LIN {X 0,Y 169.757,Z 359.407,A -85,B 0,C 180,E1 -24314.383,E2 -24314.383} C_VEL
LIN {X 0,Y 171.673,Z 362.24,A -85,B 0,C 180,E1 -24317.881,E2 -24317.881} C_VEL
LIN {X 0,Y 173.959,Z 366.587,A -85,B 0,C 180,E1 -24321.693,E2 -24321.693} C_VEL
LIN {X 0,Y 175.875,Z 371.204,A -85,B 0,C 180,E1 -24324.809,E2 -24324.809} C_VEL
LIN {X 0,Y 178.078,Z 377.199,A -85,B 0,C 180,E1 -24328.268,E2 -24328.268} C_VEL
LIN {X 0,Y 180.166,Z 384.263,A -85,B 0,C 180,E1 -24331.777,E2 -24331.777} C_VEL
LIN {X 0,Y 181.644,Z 391.259,A -85,B 0,C 180,E1 -24334.834,E2 -24334.834} C_VEL
LIN {X 0,Y 182.181,Z 398.088,A -85,B 0,C 180,E1 -24337.415,E2 -24337.415} C_VEL
LIN {X 0,Y 181.912,Z 406.288,A -85,B 0,C 180,E1 -24340.272,E2 -24340.272} C_VEL
LIN {X 0,Y 181.211,Z 412.853,A -85,B 0,C 180,E1 -24342.535,E2 -24342.535} C_VEL
LIN {X 0,Y 174.963,Z 424.329,A -85,B 0,C 180,E1 -24345.338,E2 -24345.338} C_VEL
LIN {X 0,Y 169.034,Z 433.988,A -85,B 0,C 180,E1 -24348.302,E2 -24348.302} C_VEL
LIN {X 0,Y 162.798,Z 443.459,A -85,B 0,C 180,E1 -24352.037,E2 -24352.037} C_VEL
LIN {X 0,Y 157.074,Z 451.345,A -85,B 0,C 180,E1 -24355.995,E2 -24355.995} C_VEL
LIN {X 0,Y 151.582,Z 458.707,A -85,B 0,C 180,E1 -24360.87,E2 -24360.87} C_VEL
LIN {X 0,Y 147.22,Z 464.545,A -85,B 0,C 180,E1 -24366.062,E2 -24366.062} C_VEL
LIN {X 0,Y 144.68,Z 468.003,A -85,B 0,C 180,E1 -24370.123,E2 -24370.123} C_VEL
LIN {X 0,Y 142.234,Z 471.501,A -85,B 0,C 180,E1 -24375.698,E2 -24375.698} C_VEL
LIN {X 0,Y 140.915,Z 473.81,A -85,B 0,C 180,E1 -24381.396,E2 -24381.396} C_VEL
LIN {X 0,Y 140.49,Z 474.982,A -85,B 0,C 180,E1 -24387.134,E2 -24387.134} C_VEL
LIN {X 0,Y 140.524,Z 475.138,A -85,B 0,C 180,E1 -24390.001,E2 -24390.001} C_VEL
LIN {X 0,Y 140.622,Z 474.567,A -85,B 0,C 180,E1 -24395.738,E2 -24395.738} C_VEL
LIN {X 0,Y 141.454,Z 472.874,A -85,B 0,C 180,E1 -24401.464,E2 -24401.464} C_VEL
LIN {X 0,Y 143.237,Z 470.018,A -85,B 0,C 180,E1 -24407.122,E2 -24407.122} C_VEL
LIN {X 0,Y 146.234,Z 465.93,A -85,B 0,C 180,E1 -24412.612,E2 -24412.612} C_VEL
LIN {X 0,Y 150.314,Z 460.511,A -85,B 0,C 180,E1 -24417.876,E2 -24417.876} C_VEL
LIN {X 0,Y 155.516,Z 453.606,A -85,B 0,C 180,E1 -24422.841,E2 -24422.841} C_VEL
LIN {X 0,Y 160.992,Z 446.187,A -85,B 0,C 180,E1 -24426.888,E2 -24426.888} C_VEL
LIN {X 0,Y 167.331,Z 436.789,A -85,B 0,C 180,E1 -24430.886,E2 -24430.886} C_VEL
LIN {X 0,Y 173.83,Z 426.501,A -85,B 0,C 180,E1 -24434.221,E2 -24434.221} C_VEL
LIN {X 0,Y 180.642,Z 414.423,A -85,B 0,C 180,E1 -24437.252,E2 -24437.252} C_VEL
LIN {X 0,Y 181.172,Z 413.358,A -85,B 0,C 180,E1 -24437.481,E2 -24437.481} C_VEL
LIN {X 0,Y 182,Z 406.758,A -85,B 0,C 180,E1 -24439.726,E2 -24439.726} C_VEL
LIN {X 0,Y 182.285,Z 398.5,A -85,B 0,C 180,E1 -24442.61,E2 -24442.61} C_VEL
LIN {X 0,Y 181.837,Z 391.881,A -85,B 0,C 180,E1 -24445.092,E2 -24445.092} C_VEL
LIN {X 0,Y 180.337,Z 384.628,A -85,B 0,C 180,E1 -24448.258,E2 -24448.258} C_VEL
LIN {X 0,Y 178.287,Z 377.521,A -85,B 0,C 180,E1 -24451.768,E2 -24451.768} C_VEL
LIN {X 0,Y 176.063,Z 371.611,A -85,B 0,C 180,E1 -24455.22,E2 -24455.22} C_VEL
LIN {X 0,Y 175.404,Z 369.704,A -85,B 0,C 180,E1 -24456.379,E2 -24456.379} C_VEL
LIN {X 0,Y 173.211,Z 365.171,A -85,B 0,C 180,E1 -24459.825,E2 -24459.825} C_VEL
LIN {X 0,Y 171.31,Z 361.373,A -85,B 0,C 180,E1 -24463.311,E2 -24463.311} C_VEL
LIN {X 0,Y 169.465,Z 358.831,A -85,B 0,C 180,E1 -24466.815,E2 -24466.815} C_VEL
LIN {X 0,Y 169.105,Z 357.631,A -85,B 0,C 180,E1 -24468.006,E2 -24468.006} C_VEL
LIN {X 0,Y 168.228,Z 356.362,A -85,B 0,C 180,E1 -24470.38,E2 -24470.38} C_VEL
LIN {X 0,Y 166.836,Z 353.651,A -85,B 0,C 180,E1 -24480,E2 -24480} C_VEL
LIN {X 0,Y 168.367,Z 356.425,A -85,B 0,C 180,E1 -24489.611,E2 -24489.611} C_VEL
LIN {X 0,Y 169.257,Z 357.771,A -85,B 0,C 180,E1 -24491.982,E2 -24491.982} C_VEL
LIN {X 0,Y 171.454,Z 361.806,A -85,B 0,C 180,E1 -24496.674,E2 -24496.674} C_VEL
LIN {X 0,Y 173.938,Z 367.665,A -85,B 0,C 180,E1 -24501.324,E2 -24501.324} C_VEL
LIN {X 0,Y 176.002,Z 373.065,A -85,B 0,C 180,E1 -24504.789,E2 -24504.789} C_VEL
LIN {X 0,Y 178.165,Z 379.305,A -85,B 0,C 180,E1 -24508.252,E2 -24508.252} C_VEL
LIN {X 0,Y 180.5,Z 387.992,A -85,B 0,C 180,E1 -24512.369,E2 -24512.369} C_VEL
LIN {X 0,Y 181.552,Z 394.131,A -85,B 0,C 180,E1 -24514.901,E2 -24514.901} C_VEL
LIN {X 0,Y 181.723,Z 401.562,A -85,B 0,C 180,E1 -24517.525,E2 -24517.525} C_VEL
LIN {X 0,Y 180.975,Z 411.224,A -85,B 0,C 180,E1 -24520.744,E2 -24520.744} C_VEL
LIN {X 0,Y 180.127,Z 416.685,A -85,B 0,C 180,E1 -24522.57,E2 -24522.57} C_VEL
LIN {X 0,Y 173.353,Z 428.826,A -85,B 0,C 180,E1 -24525.625,E2 -24525.625} C_VEL
LIN {X 0,Y 166.49,Z 439.624,A -85,B 0,C 180,E1 -24529.133,E2 -24529.133} C_VEL
LIN {X 0,Y 161.303,Z 447.41,A -85,B 0,C 180,E1 -24532.411,E2 -24532.411} C_VEL
LIN {X 0,Y 155.698,Z 455.072,A -85,B 0,C 180,E1 -24536.43,E2 -24536.43} C_VEL
LIN {X 0,Y 150.975,Z 461.425,A -85,B 0,C 180,E1 -24540.739,E2 -24540.739} C_VEL
LIN {X 0,Y 146.516,Z 467.472,A -85,B 0,C 180,E1 -24546.186,E2 -24546.186} C_VEL
LIN {X 0,Y 144.269,Z 470.742,A -85,B 0,C 180,E1 -24550.061,E2 -24550.061} C_VEL
LIN {X 0,Y 141.914,Z 474.25,A -85,B 0,C 180,E1 -24555.663,E2 -24555.663} C_VEL
LIN {X 0,Y 140.749,Z 476.558,A -85,B 0,C 180,E1 -24561.384,E2 -24561.384} C_VEL
LIN {X 0,Y 140.428,Z 477.718,A -85,B 0,C 180,E1 -24567.13,E2 -24567.13} C_VEL
LIN {X 0,Y 140.484,Z 477.87,A -85,B 0,C 180,E1 -24569.999,E2 -24569.999} C_VEL
LIN {X 0,Y 140.527,Z 477.263,A -85,B 0,C 180,E1 -24575.739,E2 -24575.739} C_VEL
LIN {X 0,Y 141.203,Z 475.511,A -85,B 0,C 180,E1 -24581.482,E2 -24581.482} C_VEL
LIN {X 0,Y 142.895,Z 472.592,A -85,B 0,C 180,E1 -24587.162,E2 -24587.162} C_VEL
LIN {X 0,Y 145.814,Z 468.44,A -85,B 0,C 180,E1 -24592.679,E2 -24592.679} C_VEL
LIN {X 0,Y 149.789,Z 462.941,A -85,B 0,C 180,E1 -24597.98,E2 -24597.98} C_VEL
LIN {X 0,Y 154.97,Z 455.948,A -85,B 0,C 180,E1 -24602.969,E2 -24602.969} C_VEL
LIN {X 0,Y 161.331,Z 447.25,A -85,B 0,C 180,E1 -24607.579,E2 -24607.579} C_VEL
LIN {X 0,Y 165.48,Z 440.973,A -85,B 0,C 180,E1 -24610.267,E2 -24610.267} C_VEL
LIN {X 0,Y 167.449,Z 437.392,A -85,B 0,C 180,E1 -24611.731,E2 -24611.731} C_VEL
LIN {X 0,Y 169.186,Z 431.423,A -85,B 0,C 180,E1 -24614.36,E2 -24614.36} C_VEL
LIN {X 0,Y 170.961,Z 425.058,A -85,B 0,C 180,E1 -24616.856,E2 -24616.856} C_VEL
LIN {X 0,Y 172.911,Z 420.844,A -85,B 0,C 180,E1 -24618.075,E2 -24618.075} C_VEL
LIN {X 0,Y 174.334,Z 418.074,A -85,B 0,C 180,E1 -24618.783,E2 -24618.783} C_VEL
LIN {X 0,Y 175.751,Z 409.777,A -85,B 0,C 180,E1 -24621.699,E2 -24621.699} C_VEL
LIN {X 0,Y 176.391,Z 401.393,A -85,B 0,C 180,E1 -24624.689,E2 -24624.689} C_VEL
LIN {X 0,Y 176.162,Z 395.787,A -85,B 0,C 180,E1 -24626.905,E2 -24626.905} C_VEL
LIN {X 0,Y 175.167,Z 389.996,A -85,B 0,C 180,E1 -24629.571,E2 -24629.571} C_VEL
LIN {X 0,Y 173.278,Z 382.443,A -85,B 0,C 180,E1 -24633.503,E2 -24633.503} C_VEL
LIN {X 0,Y 171.498,Z 376.48,A -85,B 0,C 180,E1 -24637.089,E2 -24637.089} C_VEL
LIN {X 0,Y 169.651,Z 371.634,A -85,B 0,C 180,E1 -24640.646,E2 -24640.646} C_VEL
LIN {X 0,Y 168.286,Z 367.78,A -85,B 0,C 180,E1 -24643.842,E2 -24643.842} C_VEL
LIN {X 0,Y 166.603,Z 364.532,A -85,B 0,C 180,E1 -24647.824,E2 -24647.824} C_VEL
LIN {X 0,Y 165.812,Z 363.028,A -85,B 0,C 180,E1 -24650.239,E2 -24650.239} C_VEL
LIN {X 0,Y 164.425,Z 359.9,A -85,B 0,C 180,E1 -24660,E2 -24660} C_VEL
LIN {X 0,Y 165.622,Z 362.919,A -85,B 0,C 180,E1 -24669.773,E2 -24669.773} C_VEL
LIN {X 0,Y 166.413,Z 364.278,A -85,B 0,C 180,E1 -24672.191,E2 -24672.191} C_VEL
LIN {X 0,Y 168.45,Z 368.116,A -85,B 0,C 180,E1 -24676.981,E2 -24676.981} C_VEL
LIN {X 0,Y 170.237,Z 371.88,A -85,B 0,C 180,E1 -24680.543,E2 -24680.543} C_VEL
LIN {X 0,Y 172.11,Z 376.812,A -85,B 0,C 180,E1 -24684.101,E2 -24684.101} C_VEL
LIN {X 0,Y 174.257,Z 383.704,A -85,B 0,C 180,E1 -24688.222,E2 -24688.222} C_VEL
LIN {X 0,Y 175.928,Z 391.102,A -85,B 0,C 180,E1 -24691.96,E2 -24691.96} C_VEL
LIN {X 0,Y 176.792,Z 396.739,A -85,B 0,C 180,E1 -24694.505,E2 -24694.505} C_VEL
LIN {X 0,Y 176.78,Z 404.047,A -85,B 0,C 180,E1 -24697.337,E2 -24697.337} C_VEL
LIN {X 0,Y 175.829,Z 412.936,A -85,B 0,C 180,E1 -24700.588,E2 -24700.588} C_VEL
LIN {X 0,Y 175.433,Z 415.028,A -85,B 0,C 180,E1 -24701.313,E2 -24701.313} C_VEL
LIN {X 0,Y 168.9,Z 426.171,A -85,B 0,C 180,E1 -24704.131,E2 -24704.131} C_VEL
LIN {X 0,Y 162.532,Z 435.96,A -85,B 0,C 180,E1 -24707.315,E2 -24707.315} C_VEL
LIN {X 0,Y 156.314,Z 444.758,A -85,B 0,C 180,E1 -24710.992,E2 -24710.992} C_VEL
LIN {X 0,Y 150.41,Z 452.421,A -85,B 0,C 180,E1 -24715.085,E2 -24715.085} C_VEL
LIN {X 0,Y 145.379,Z 458.777,A -85,B 0,C 180,E1 -24719.498,E2 -24719.498} C_VEL
LIN {X 0,Y 140.723,Z 464.616,A -85,B 0,C 180,E1 -24724.882,E2 -24724.882} C_VEL
LIN {X 0,Y 137.979,Z 468.074,A -85,B 0,C 180,E1 -24729.113,E2 -24729.113} C_VEL
LIN {X 0,Y 135.333,Z 471.571,A -85,B 0,C 180,E1 -24734.952,E2 -24734.952} C_VEL
LIN {X 0,Y 133.879,Z 473.879,A -85,B 0,C 180,E1 -24740.94,E2 -24740.94} C_VEL
LIN {X 0,Y 133.402,Z 475.051,A -85,B 0,C 180,E1 -24746.981,E2 -24746.981} C_VEL
LIN {X 0,Y 133.449,Z 475.206,A -85,B 0,C 180,E1 -24750.001,E2 -24750.001} C_VEL
LIN {X 0,Y 133.549,Z 474.636,A -85,B 0,C 180,E1 -24756.043,E2 -24756.043} C_VEL
LIN {X 0,Y 134.476,Z 472.943,A -85,B 0,C 180,E1 -24762.068,E2 -24762.068} C_VEL
LIN {X 0,Y 136.423,Z 470.087,A -85,B 0,C 180,E1 -24768.006,E2 -24768.006} C_VEL
LIN {X 0,Y 139.649,Z 465.998,A -85,B 0,C 180,E1 -24773.742,E2 -24773.742} C_VEL
LIN {X 0,Y 144.034,Z 460.579,A -85,B 0,C 180,E1 -24779.206,E2 -24779.206} C_VEL
LIN {X 0,Y 149.555,Z 453.674,A -85,B 0,C 180,E1 -24784.328,E2 -24784.328} C_VEL
LIN {X 0,Y 155.35,Z 446.254,A -85,B 0,C 180,E1 -24788.466,E2 -24788.466} C_VEL
LIN {X 0,Y 161.635,Z 437.367,A -85,B 0,C 180,E1 -24792.339,E2 -24792.339} C_VEL
LIN {X 0,Y 167.728,Z 428.192,A -85,B 0,C 180,E1 -24795.425,E2 -24795.425} C_VEL
LIN {X 0,Y 174.184,Z 417.434,A -85,B 0,C 180,E1 -24798.283,E2 -24798.283} C_VEL
LIN {X 0,Y 175.709,Z 414.491,A -85,B 0,C 180,E1 -24799.022,E2 -24799.022} C_VEL
LIN {X 0,Y 176.745,Z 406.401,A -85,B 0,C 180,E1 -24801.952,E2 -24801.952} C_VEL
LIN {X 0,Y 176.961,Z 398.81,A -85,B 0,C 180,E1 -24804.839,E2 -24804.839} C_VEL
LIN {X 0,Y 176.605,Z 394.429,A -85,B 0,C 180,E1 -24806.688,E2 -24806.688} C_VEL
LIN {X 0,Y 175.597,Z 388.83,A -85,B 0,C 180,E1 -24809.343,E2 -24809.343} C_VEL
LIN {X 0,Y 174.037,Z 382.495,A -85,B 0,C 180,E1 -24812.674,E2 -24812.674} C_VEL
LIN {X 0,Y 171.903,Z 375.917,A -85,B 0,C 180,E1 -24816.756,E2 -24816.756} C_VEL
LIN {X 0,Y 170.434,Z 372.256,A -85,B 0,C 180,E1 -24819.482,E2 -24819.482} C_VEL
LIN {X 0,Y 168.363,Z 367.695,A -85,B 0,C 180,E1 -24823.759,E2 -24823.759} C_VEL
LIN {X 0,Y 165.864,Z 363.18,A -85,B 0,C 180,E1 -24830.242,E2 -24830.242} C_VEL
LIN {X 0,Y 164.581,Z 360.396,A -85,B 0,C 180,E1 -24840,E2 -24840} C_VEL
LIN {X 0,Y 166.021,Z 363.258,A -85,B 0,C 180,E1 -24849.748,E2 -24849.748} C_VEL
LIN {X 0,Y 167.674,Z 366.823,A -85,B 0,C 180,E1 -24854.565,E2 -24854.565} C_VEL
LIN {X 0,Y 168.747,Z 369.117,A -85,B 0,C 180,E1 -24856.95,E2 -24856.95} C_VEL
LIN {X 0,Y 170.421,Z 373.342,A -85,B 0,C 180,E1 -24860.52,E2 -24860.52} C_VEL
LIN {X 0,Y 172.193,Z 378.663,A -85,B 0,C 180,E1 -24864.088,E2 -24864.088} C_VEL
LIN {X 0,Y 174.193,Z 385.479,A -85,B 0,C 180,E1 -24868.019,E2 -24868.019} C_VEL
LIN {X 0,Y 175.904,Z 393.489,A -85,B 0,C 180,E1 -24871.964,E2 -24871.964} C_VEL
LIN {X 0,Y 176.51,Z 399.127,A -85,B 0,C 180,E1 -24874.359,E2 -24874.359} C_VEL
LIN {X 0,Y 176.286,Z 405.559,A -85,B 0,C 180,E1 -24876.727,E2 -24876.727} C_VEL
LIN {X 0,Y 175.355,Z 413.475,A -85,B 0,C 180,E1 -24879.548,E2 -24879.548} C_VEL
LIN {X 0,Y 174.46,Z 418.22,A -85,B 0,C 180,E1 -24881.212,E2 -24881.212} C_VEL
LIN {X 0,Y 168.31,Z 428.759,A -85,B 0,C 180,E1 -24883.921,E2 -24883.921} C_VEL
LIN {X 0,Y 161.156,Z 439.556,A -85,B 0,C 180,E1 -24887.471,E2 -24887.471} C_VEL
LIN {X 0,Y 155.66,Z 447.341,A -85,B 0,C 180,E1 -24890.795,E2 -24890.795} C_VEL
LIN {X 0,Y 149.794,Z 455.004,A -85,B 0,C 180,E1 -24894.918,E2 -24894.918} C_VEL
LIN {X 0,Y 144.763,Z 461.356,A -85,B 0,C 180,E1 -24899.352,E2 -24899.352} C_VEL
LIN {X 0,Y 140.585,Z 466.634,A -85,B 0,C 180,E1 -24904.136,E2 -24904.136} C_VEL
LIN {X 0,Y 137.547,Z 470.673,A -85,B 0,C 180,E1 -24909.042,E2 -24909.042} C_VEL
LIN {X 0,Y 134.985,Z 474.181,A -85,B 0,C 180,E1 -24914.91,E2 -24914.91} C_VEL
LIN {X 0,Y 133.702,Z 476.489,A -85,B 0,C 180,E1 -24920.926,E2 -24920.926} C_VEL
LIN {X 0,Y 133.33,Z 477.649,A -85,B 0,C 180,E1 -24926.977,E2 -24926.977} C_VEL
LIN {X 0,Y 133.39,Z 477.801,A -85,B 0,C 180,E1 -24929.999,E2 -24929.999} C_VEL
LIN {X 0,Y 133.443,Z 477.193,A -85,B 0,C 180,E1 -24936.045,E2 -24936.045} C_VEL
LIN {X 0,Y 134.215,Z 475.441,A -85,B 0,C 180,E1 -24942.089,E2 -24942.089} C_VEL
LIN {X 0,Y 136.089,Z 472.522,A -85,B 0,C 180,E1 -24948.049,E2 -24948.049} C_VEL
LIN {X 0,Y 139.236,Z 468.369,A -85,B 0,C 180,E1 -24953.814,E2 -24953.814} C_VEL
LIN {X 0,Y 143.498,Z 462.87,A -85,B 0,C 180,E1 -24959.323,E2 -24959.323} C_VEL
LIN {X 0,Y 149,Z 455.877,A -85,B 0,C 180,E1 -24964.471,E2 -24964.471} C_VEL
LIN {X 0,Y 154.858,Z 448.4,A -85,B 0,C 180,E1 -24968.609,E2 -24968.609} C_VEL
LIN {X 0,Y 160.21,Z 440.736,A -85,B 0,C 180,E1 -24971.986,E2 -24971.986} C_VEL
LIN {X 0,Y 167.239,Z 430.174,A -85,B 0,C 180,E1 -24975.592,E2 -24975.592} C_VEL
LIN {X 0,Y 172.911,Z 420.844,A -85,B 0,C 180,E1 -24978.075,E2 -24978.075} C_VEL
LIN {X 0,Y 174.029,Z 418.111,A -85,B 0,C 180,E1 -24978.879,E2 -24978.879} C_VEL
LIN {X 0,Y 174.314,Z 414.412,A -85,B 0,C 180,E1 -24980.374,E2 -24980.374} C_VEL
LIN {X 0,Y 173.58,Z 411.263,A -85,B 0,C 180,E1 -24982.025,E2 -24982.025} C_VEL
LIN {X 0,Y 171.428,Z 404.974,A -85,B 0,C 180,E1 -24985.6,E2 -24985.6} C_VEL
LIN {X 0,Y 171.221,Z 402.477,A -85,B 0,C 180,E1 -24986.724,E2 -24986.724} C_VEL
LIN {X 0,Y 170.872,Z 397.357,A -85,B 0,C 180,E1 -24989.063,E2 -24989.063} C_VEL
LIN {X 0,Y 169.337,Z 388.941,A -85,B 0,C 180,E1 -24993.503,E2 -24993.503} C_VEL
LIN {X 0,Y 167.609,Z 382.016,A -85,B 0,C 180,E1 -24997.829,E2 -24997.829} C_VEL
LIN {X 0,Y 166.093,Z 377.299,A -85,B 0,C 180,E1 -25001.497,E2 -25001.497} C_VEL
LIN {X 0,Y 164.727,Z 373.352,A -85,B 0,C 180,E1 -25005.168,E2 -25005.168} C_VEL
LIN {X 0,Y 163.19,Z 369.785,A -85,B 0,C 180,E1 -25010.081,E2 -25010.081} C_VEL
LIN {X 0,Y 161.909,Z 366.583,A -85,B 0,C 180,E1 -25020,E2 -25020} C_VEL
LIN {X 0,Y 162.994,Z 369.639,A -85,B 0,C 180,E1 -25029.932,E2 -25029.932} C_VEL
LIN {X 0,Y 163.677,Z 371.126,A -85,B 0,C 180,E1 -25032.398,E2 -25032.398} C_VEL
LIN {X 0,Y 165.526,Z 375.076,A -85,B 0,C 180,E1 -25037.29,E2 -25037.29} C_VEL
LIN {X 0,Y 167.091,Z 379.052,A -85,B 0,C 180,E1 -25040.948,E2 -25040.948} C_VEL
LIN {X 0,Y 168.387,Z 383.002,A -85,B 0,C 180,E1 -25043.845,E2 -25043.845} C_VEL
LIN {X 0,Y 169.988,Z 389.297,A -85,B 0,C 180,E1 -25047.74,E2 -25047.74} C_VEL
LIN {X 0,Y 171.246,Z 396.493,A -85,B 0,C 180,E1 -25051.551,E2 -25051.551} C_VEL
LIN {X 0,Y 171.666,Z 402.352,A -85,B 0,C 180,E1 -25054.252,E2 -25054.252} C_VEL
LIN {X 0,Y 171.186,Z 409.165,A -85,B 0,C 180,E1 -25056.995,E2 -25056.995} C_VEL
LIN {X 0,Y 170.125,Z 415.788,A -85,B 0,C 180,E1 -25059.562,E2 -25059.562} C_VEL
LIN {X 0,Y 169.643,Z 417.048,A -85,B 0,C 180,E1 -25059.969,E2 -25059.969} C_VEL
LIN {X 0,Y 162.898,Z 427.877,A -85,B 0,C 180,E1 -25062.827,E2 -25062.827} C_VEL
LIN {X 0,Y 155.914,Z 438.002,A -85,B 0,C 180,E1 -25066.307,E2 -25066.307} C_VEL
LIN {X 0,Y 149.904,Z 446.048,A -85,B 0,C 180,E1 -25069.863,E2 -25069.863} C_VEL
LIN {X 0,Y 143.789,Z 453.497,A -85,B 0,C 180,E1 -25074.091,E2 -25074.091} C_VEL
LIN {X 0,Y 137.913,Z 460.456,A -85,B 0,C 180,E1 -25079.365,E2 -25079.365} C_VEL
LIN {X 0,Y 133.197,Z 465.923,A -85,B 0,C 180,E1 -25085.034,E2 -25085.034} C_VEL
LIN {X 0,Y 129.681,Z 470.047,A -85,B 0,C 180,E1 -25091.026,E2 -25091.026} C_VEL
LIN {X 0,Y 127.536,Z 472.939,A -85,B 0,C 180,E1 -25097.267,E2 -25097.267} C_VEL
LIN {X 0,Y 126.472,Z 474.674,A -85,B 0,C 180,E1 -25103.62,E2 -25103.62} C_VEL
LIN {X 0,Y 126.36,Z 475.275,A -85,B 0,C 180,E1 -25110.001,E2 -25110.001} C_VEL
LIN {X 0,Y 126.472,Z 474.705,A -85,B 0,C 180,E1 -25116.382,E2 -25116.382} C_VEL
LIN {X 0,Y 127.509,Z 473.012,A -85,B 0,C 180,E1 -25122.738,E2 -25122.738} C_VEL
LIN {X 0,Y 129.645,Z 470.156,A -85,B 0,C 180,E1 -25128.982,E2 -25128.982} C_VEL
LIN {X 0,Y 133.132,Z 466.067,A -85,B 0,C 180,E1 -25134.982,E2 -25134.982} C_VEL
LIN {X 0,Y 137.832,Z 460.647,A -85,B 0,C 180,E1 -25140.658,E2 -25140.658} C_VEL
LIN {X 0,Y 143.718,Z 453.742,A -85,B 0,C 180,E1 -25145.932,E2 -25145.932} C_VEL
LIN {X 0,Y 149.832,Z 446.322,A -85,B 0,C 180,E1 -25150.163,E2 -25150.163} C_VEL
LIN {X 0,Y 156.768,Z 436.984,A -85,B 0,C 180,E1 -25154.279,E2 -25154.279} C_VEL
LIN {X 0,Y 163.913,Z 426.634,A -85,B 0,C 180,E1 -25157.699,E2 -25157.699} C_VEL
LIN {X 0,Y 170.18,Z 416.179,A -85,B 0,C 180,E1 -25160.445,E2 -25160.445} C_VEL
LIN {X 0,Y 171.391,Z 408.308,A -85,B 0,C 180,E1 -25163.518,E2 -25163.518} C_VEL
LIN {X 0,Y 171.779,Z 400.794,A -85,B 0,C 180,E1 -25166.575,E2 -25166.575} C_VEL
LIN {X 0,Y 171.063,Z 394.524,A -85,B 0,C 180,E1 -25169.629,E2 -25169.629} C_VEL
LIN {X 0,Y 169.662,Z 387.414,A -85,B 0,C 180,E1 -25173.557,E2 -25173.557} C_VEL
LIN {X 0,Y 167.843,Z 380.947,A -85,B 0,C 180,E1 -25177.861,E2 -25177.861} C_VEL
LIN {X 0,Y 166.224,Z 376.665,A -85,B 0,C 180,E1 -25181.512,E2 -25181.512} C_VEL
LIN {X 0,Y 165.447,Z 374.67,A -85,B 0,C 180,E1 -25183.464,E2 -25183.464} C_VEL
LIN {X 0,Y 163.204,Z 369.95,A -85,B 0,C 180,E1 -25190.081,E2 -25190.081} C_VEL
LIN {X 0,Y 161.931,Z 367.699,A -85,B 0,C 180,E1 -25197.512,E2 -25197.512} C_VEL
LIN {X 0,Y 162.05,Z 367.06,A -85,B 0,C 180,E1 -25200,E2 -25200} C_VEL
LIN {X 0,Y 162.69,Z 369.111,A -85,B 0,C 180,E1 -25207.446,E2 -25207.446} C_VEL
LIN {X 0,Y 163.375,Z 370.052,A -85,B 0,C 180,E1 -25209.908,E2 -25209.908} C_VEL
LIN {X 0,Y 164.872,Z 373.683,A -85,B 0,C 180,E1 -25214.818,E2 -25214.818} C_VEL
LIN {X 0,Y 166.248,Z 377.555,A -85,B 0,C 180,E1 -25218.485,E2 -25218.485} C_VEL
LIN {X 0,Y 167.743,Z 382.291,A -85,B 0,C 180,E1 -25222.152,E2 -25222.152} C_VEL
LIN {X 0,Y 169.21,Z 388.112,A -85,B 0,C 180,E1 -25225.856,E2 -25225.856} C_VEL
LIN {X 0,Y 170.577,Z 394.97,A -85,B 0,C 180,E1 -25229.631,E2 -25229.631} C_VEL
LIN {X 0,Y 171.269,Z 400.296,A -85,B 0,C 180,E1 -25232.239,E2 -25232.239} C_VEL
LIN {X 0,Y 171.155,Z 406.466,A -85,B 0,C 180,E1 -25234.79,E2 -25234.79} C_VEL
LIN {X 0,Y 169.762,Z 416.035,A -85,B 0,C 180,E1 -25238.388,E2 -25238.388} C_VEL
LIN {X 0,Y 168.754,Z 420.109,A -85,B 0,C 180,E1 -25239.888,E2 -25239.888} C_VEL
LIN {X 0,Y 162.345,Z 430.322,A -85,B 0,C 180,E1 -25242.613,E2 -25242.613} C_VEL
LIN {X 0,Y 154.932,Z 440.845,A -85,B 0,C 180,E1 -25246.229,E2 -25246.229} C_VEL
LIN {X 0,Y 149.286,Z 448.484,A -85,B 0,C 180,E1 -25249.66,E2 -25249.66} C_VEL
LIN {X 0,Y 143.161,Z 455.946,A -85,B 0,C 180,E1 -25253.906,E2 -25253.906} C_VEL
LIN {X 0,Y 137.282,Z 462.904,A -85,B 0,C 180,E1 -25259.206,E2 -25259.206} C_VEL
LIN {X 0,Y 132.68,Z 468.375,A -85,B 0,C 180,E1 -25264.927,E2 -25264.927} C_VEL
LIN {X 0,Y 129.322,Z 472.512,A -85,B 0,C 180,E1 -25270.969,E2 -25270.969} C_VEL
LIN {X 0,Y 127.253,Z 475.412,A -85,B 0,C 180,E1 -25277.236,E2 -25277.236} C_VEL
LIN {X 0,Y 126.366,Z 477.142,A -85,B 0,C 180,E1 -25283.613,E2 -25283.613} C_VEL
LIN {X 0,Y 126.307,Z 477.733,A -85,B 0,C 180,E1 -25289.999,E2 -25289.999} C_VEL
LIN {X 0,Y 126.366,Z 477.124,A -85,B 0,C 180,E1 -25296.385,E2 -25296.385} C_VEL
LIN {X 0,Y 127.252,Z 475.371,A -85,B 0,C 180,E1 -25302.761,E2 -25302.761} C_VEL
LIN {X 0,Y 129.322,Z 472.452,A -85,B 0,C 180,E1 -25309.029,E2 -25309.029} C_VEL
LIN {X 0,Y 132.695,Z 468.299,A -85,B 0,C 180,E1 -25315.067,E2 -25315.067} C_VEL
LIN {X 0,Y 137.287,Z 462.799,A -85,B 0,C 180,E1 -25320.79,E2 -25320.79} C_VEL
LIN {X 0,Y 143.153,Z 455.806,A -85,B 0,C 180,E1 -25326.094,E2 -25326.094} C_VEL
LIN {X 0,Y 149.323,Z 448.329,A -85,B 0,C 180,E1 -25330.325,E2 -25330.325} C_VEL
LIN {X 0,Y 155.968,Z 439.309,A -85,B 0,C 180,E1 -25334.299,E2 -25334.299} C_VEL
LIN {X 0,Y 163.422,Z 428.466,A -85,B 0,C 180,E1 -25337.886,E2 -25337.886} C_VEL
LIN {X 0,Y 168.668,Z 419.941,A -85,B 0,C 180,E1 -25340.099,E2 -25340.099} C_VEL
LIN {X 0,Y 170.195,Z 412.669,A -85,B 0,C 180,E1 -25342.802,E2 -25342.802} C_VEL
LIN {X 0,Y 171.177,Z 404.643,A -85,B 0,C 180,E1 -25345.854,E2 -25345.854} C_VEL
LIN {X 0,Y 171.221,Z 402.477,A -85,B 0,C 180,E1 -25346.724,E2 -25346.724} C_VEL
LIN {X 0,Y 170.972,Z 400.224,A -85,B 0,C 180,E1 -25347.793,E2 -25347.793} C_VEL
LIN {X 0,Y 169.819,Z 397.655,A -85,B 0,C 180,E1 -25349.539,E2 -25349.539} C_VEL
LIN {X 0,Y 166.964,Z 394.628,A -85,B 0,C 180,E1 -25352.65,E2 -25352.65} C_VEL
LIN {X 0,Y 164.514,Z 391.376,A -85,B 0,C 180,E1 -25355.875,E2 -25355.875} C_VEL
LIN {X 0,Y 164.23,Z 390.509,A -85,B 0,C 180,E1 -25356.508,E2 -25356.508} C_VEL
LIN {X 0,Y 163.59,Z 387.437,A -85,B 0,C 180,E1 -25358.582,E2 -25358.582} C_VEL
LIN {X 0,Y 162.357,Z 382.857,A -85,B 0,C 180,E1 -25362.362,E2 -25362.362} C_VEL
LIN {X 0,Y 161.244,Z 379.091,A -85,B 0,C 180,E1 -25366.13,E2 -25366.13} C_VEL
LIN {X 0,Y 160.263,Z 376.484,A -85,B 0,C 180,E1 -25369.898,E2 -25369.898} C_VEL
LIN {X 0,Y 159.127,Z 374.71,A -85,B 0,C 180,E1 -25374.933,E2 -25374.933} C_VEL
LIN {X 0,Y 159.122,Z 373.166,A -85,B 0,C 180,E1 -25380,E2 -25380} C_VEL
LIN {X 0,Y 160.082,Z 376.275,A -85,B 0,C 180,E1 -25390.114,E2 -25390.114} C_VEL
LIN {X 0,Y 161.438,Z 379.668,A -85,B 0,C 180,E1 -25395.142,E2 -25395.142} C_VEL
LIN {X 0,Y 162.803,Z 383.124,A -85,B 0,C 180,E1 -25398.89,E2 -25398.89} C_VEL
LIN {X 0,Y 163.686,Z 386.005,A -85,B 0,C 180,E1 -25401.405,E2 -25401.405} C_VEL
LIN {X 0,Y 164.907,Z 391.468,A -85,B 0,C 180,E1 -25405.226,E2 -25405.226} C_VEL
LIN {X 0,Y 165.966,Z 398.018,A -85,B 0,C 180,E1 -25409.143,E2 -25409.143} C_VEL
LIN {X 0,Y 166.457,Z 404.232,A -85,B 0,C 180,E1 -25412.393,E2 -25412.393} C_VEL
LIN {X 0,Y 165.964,Z 410.46,A -85,B 0,C 180,E1 -25415.137,E2 -25415.137} C_VEL
LIN {X 0,Y 164.599,Z 417.805,A -85,B 0,C 180,E1 -25418.174,E2 -25418.174} C_VEL
LIN {X 0,Y 159.304,Z 426.315,A -85,B 0,C 180,E1 -25420.449,E2 -25420.449} C_VEL
LIN {X 0,Y 152.612,Z 435.727,A -85,B 0,C 180,E1 -25423.534,E2 -25423.534} C_VEL
LIN {X 0,Y 145.495,Z 444.901,A -85,B 0,C 180,E1 -25427.45,E2 -25427.45} C_VEL
LIN {X 0,Y 138.93,Z 452.563,A -85,B 0,C 180,E1 -25431.709,E2 -25431.709} C_VEL
LIN {X 0,Y 133.256,Z 458.919,A -85,B 0,C 180,E1 -25436.376,E2 -25436.376} C_VEL
LIN {X 0,Y 127.915,Z 464.757,A -85,B 0,C 180,E1 -25442.161,E2 -25442.161} C_VEL
LIN {X 0,Y 124.741,Z 468.214,A -85,B 0,C 180,E1 -25446.774,E2 -25446.774} C_VEL
LIN {X 0,Y 121.61,Z 471.711,A -85,B 0,C 180,E1 -25453.206,E2 -25453.206} C_VEL
LIN {X 0,Y 119.847,Z 474.018,A -85,B 0,C 180,E1 -25459.869,E2 -25459.869} C_VEL
LIN {X 0,Y 119.225,Z 475.189,A -85,B 0,C 180,E1 -25466.622,E2 -25466.622} C_VEL
LIN {X 0,Y 119.279,Z 475.344,A -85,B 0,C 180,E1 -25470.001,E2 -25470.001} C_VEL
LIN {X 0,Y 119.42,Z 474.774,A -85,B 0,C 180,E1 -25476.761,E2 -25476.761} C_VEL
LIN {X 0,Y 120.556,Z 473.081,A -85,B 0,C 180,E1 -25483.486,E2 -25483.486} C_VEL
LIN {X 0,Y 122.913,Z 470.225,A -85,B 0,C 180,E1 -25490.065,E2 -25490.065} C_VEL
LIN {X 0,Y 126.687,Z 466.135,A -85,B 0,C 180,E1 -25496.348,E2 -25496.348} C_VEL
LIN {X 0,Y 131.719,Z 460.715,A -85,B 0,C 180,E1 -25502.247,E2 -25502.247} C_VEL
LIN {X 0,Y 137.991,Z 453.809,A -85,B 0,C 180,E1 -25507.675,E2 -25507.675} C_VEL
LIN {X 0,Y 144.455,Z 446.389,A -85,B 0,C 180,E1 -25511.988,E2 -25511.988} C_VEL
LIN {X 0,Y 151.321,Z 437.576,A -85,B 0,C 180,E1 -25515.954,E2 -25515.954} C_VEL
LIN {X 0,Y 158.045,Z 428.325,A -85,B 0,C 180,E1 -25519.11,E2 -25519.11} C_VEL
LIN {X 0,Y 164.635,Z 418.192,A -85,B 0,C 180,E1 -25521.842,E2 -25521.842} C_VEL
LIN {X 0,Y 166.18,Z 409.817,A -85,B 0,C 180,E1 -25525.318,E2 -25525.318} C_VEL
LIN {X 0,Y 166.578,Z 403.469,A -85,B 0,C 180,E1 -25528.17,E2 -25528.17} C_VEL
LIN {X 0,Y 165.962,Z 397.19,A -85,B 0,C 180,E1 -25531.549,E2 -25531.549} C_VEL
LIN {X 0,Y 164.868,Z 390.771,A -85,B 0,C 180,E1 -25535.483,E2 -25535.483} C_VEL
LIN {X 0,Y 163.84,Z 386.388,A -85,B 0,C 180,E1 -25538.616,E2 -25538.616} C_VEL
LIN {X 0,Y 162.508,Z 382.25,A -85,B 0,C 180,E1 -25542.378,E2 -25542.378} C_VEL
LIN {X 0,Y 161.638,Z 379.985,A -85,B 0,C 180,E1 -25544.877,E2 -25544.877} C_VEL
LIN {X 0,Y 160.269,Z 376.605,A -85,B 0,C 180,E1 -25549.897,E2 -25549.897} C_VEL
LIN {X 0,Y 159.239,Z 374.931,A -85,B 0,C 180,E1 -25554.936,E2 -25554.936} C_VEL
LIN {X 0,Y 159.253,Z 373.617,A -85,B 0,C 180,E1 -25560,E2 -25560} C_VEL
LIN {X 0,Y 159.83,Z 375.658,A -85,B 0,C 180,E1 -25567.58,E2 -25567.58} C_VEL
LIN {X 0,Y 160.442,Z 376.752,A -85,B 0,C 180,E1 -25570.091,E2 -25570.091} C_VEL
LIN {X 0,Y 161.799,Z 380.402,A -85,B 0,C 180,E1 -25575.107,E2 -25575.107} C_VEL
LIN {X 0,Y 162.95,Z 384.468,A -85,B 0,C 180,E1 -25578.872,E2 -25578.872} C_VEL
LIN {X 0,Y 164.465,Z 391.035,A -85,B 0,C 180,E1 -25583.701,E2 -25583.701} C_VEL
LIN {X 0,Y 165.579,Z 397.873,A -85,B 0,C 180,E1 -25587.833,E2 -25587.833} C_VEL
LIN {X 0,Y 166.195,Z 404.025,A -85,B 0,C 180,E1 -25591.112,E2 -25591.112} C_VEL
LIN {X 0,Y 165.896,Z 409.198,A -85,B 0,C 180,E1 -25593.417,E2 -25593.417} C_VEL
LIN {X 0,Y 164.266,Z 418.104,A -85,B 0,C 180,E1 -25596.987,E2 -25596.987} C_VEL
LIN {X 0,Y 163.051,Z 422.048,A -85,B 0,C 180,E1 -25598.457,E2 -25598.457} C_VEL
LIN {X 0,Y 155.314,Z 433.512,A -85,B 0,C 180,E1 -25601.7,E2 -25601.7} C_VEL
LIN {X 0,Y 147.986,Z 443.183,A -85,B 0,C 180,E1 -25605.318,E2 -25605.318} C_VEL
LIN {X 0,Y 141.086,Z 451.774,A -85,B 0,C 180,E1 -25609.64,E2 -25609.64} C_VEL
LIN {X 0,Y 135.794,Z 457.742,A -85,B 0,C 180,E1 -25613.474,E2 -25613.474} C_VEL
LIN {X 0,Y 129.808,Z 464.318,A -85,B 0,C 180,E1 -25619.045,E2 -25619.045} C_VEL
LIN {X 0,Y 125.197,Z 469.464,A -85,B 0,C 180,E1 -25625.1,E2 -25625.1} C_VEL
LIN {X 0,Y 122.595,Z 472.443,A -85,B 0,C 180,E1 -25629.881,E2 -25629.881} C_VEL
LIN {X 0,Y 120.279,Z 475.343,A -85,B 0,C 180,E1 -25636.483,E2 -25636.483} C_VEL
LIN {X 0,Y 119.279,Z 477.073,A -85,B 0,C 180,E1 -25643.231,E2 -25643.231} C_VEL
LIN {X 0,Y 119.226,Z 477.664,A -85,B 0,C 180,E1 -25649.999,E2 -25649.999} C_VEL
LIN {X 0,Y 119.279,Z 477.054,A -85,B 0,C 180,E1 -25656.766,E2 -25656.766} C_VEL
LIN {X 0,Y 120.278,Z 475.301,A -85,B 0,C 180,E1 -25663.515,E2 -25663.515} C_VEL
LIN {X 0,Y 122.596,Z 472.382,A -85,B 0,C 180,E1 -25670.117,E2 -25670.117} C_VEL
LIN {X 0,Y 126.228,Z 468.228,A -85,B 0,C 180,E1 -25676.448,E2 -25676.448} C_VEL
LIN {X 0,Y 131.176,Z 462.728,A -85,B 0,C 180,E1 -25682.394,E2 -25682.394} C_VEL
LIN {X 0,Y 137.435,Z 455.735,A -85,B 0,C 180,E1 -25687.851,E2 -25687.851} C_VEL
LIN {X 0,Y 143.922,Z 448.257,A -85,B 0,C 180,E1 -25692.176,E2 -25692.176} C_VEL
LIN {X 0,Y 150.923,Z 439.237,A -85,B 0,C 180,E1 -25696.199,E2 -25696.199} C_VEL
LIN {X 0,Y 158.73,Z 428.394,A -85,B 0,C 180,E1 -25699.795,E2 -25699.795} C_VEL
LIN {X 0,Y 163.028,Z 421.821,A -85,B 0,C 180,E1 -25701.529,E2 -25701.529} C_VEL
LIN {X 0,Y 164.539,Z 416.295,A -85,B 0,C 180,E1 -25703.662,E2 -25703.662} C_VEL
LIN {X 0,Y 165.798,Z 409.022,A -85,B 0,C 180,E1 -25706.561,E2 -25706.561} C_VEL
LIN {X 0,Y 166.05,Z 403.657,A -85,B 0,C 180,E1 -25708.969,E2 -25708.969} C_VEL
LIN {X 0,Y 165.454,Z 397.687,A -85,B 0,C 180,E1 -25712.145,E2 -25712.145} C_VEL
LIN {X 0,Y 164.535,Z 391.769,A -85,B 0,C 180,E1 -25715.631,E2 -25715.631} C_VEL
LIN {X 0,Y 164.23,Z 390.509,A -85,B 0,C 180,E1 -25716.508,E2 -25716.508} C_VEL
LIN {X 0,Y 163.221,Z 388.4,A -85,B 0,C 180,E1 -25718.405,E2 -25718.405} C_VEL
LIN {X 0,Y 161.798,Z 387.179,A -85,B 0,C 180,E1 -25720.393,E2 -25720.393} C_VEL
LIN {X 0,Y 158.053,Z 385.354,A -85,B 0,C 180,E1 -25725.964,E2 -25725.964} C_VEL
LIN {X 0,Y 157.534,Z 384.575,A -85,B 0,C 180,E1 -25727.387,E2 -25727.387} C_VEL
LIN {X 0,Y 156.992,Z 382.853,A -85,B 0,C 180,E1 -25730.007,E2 -25730.007} C_VEL
LIN {X 0,Y 156.038,Z 381.122,A -85,B 0,C 180,E1 -25734.832,E2 -25734.832} C_VEL
LIN {X 0,Y 156.082,Z 379.61,A -85,B 0,C 180,E1 -25740,E2 -25740} C_VEL
LIN {X 0,Y 156.653,Z 382.302,A -85,B 0,C 180,E1 -25749.262,E2 -25749.262} C_VEL
LIN {X 0,Y 157.387,Z 384.427,A -85,B 0,C 180,E1 -25752.902,E2 -25752.902} C_VEL
LIN {X 0,Y 158.593,Z 387.947,A -85,B 0,C 180,E1 -25757.334,E2 -25757.334} C_VEL
LIN {X 0,Y 159.57,Z 391.361,A -85,B 0,C 180,E1 -25760.631,E2 -25760.631} C_VEL
LIN {X 0,Y 160.478,Z 396.731,A -85,B 0,C 180,E1 -25764.585,E2 -25764.585} C_VEL
LIN {X 0,Y 161.148,Z 403.235,A -85,B 0,C 180,E1 -25768.668,E2 -25768.668} C_VEL
LIN {X 0,Y 161.269,Z 408.415,A -85,B 0,C 180,E1 -25771.531,E2 -25771.531} C_VEL
LIN {X 0,Y 160.491,Z 414.089,A -85,B 0,C 180,E1 -25774.172,E2 -25774.172} C_VEL
LIN {X 0,Y 159.139,Z 419.845,A -85,B 0,C 180,E1 -25776.683,E2 -25776.683} C_VEL
LIN {X 0,Y 152.383,Z 429.645,A -85,B 0,C 180,E1 -25779.422,E2 -25779.422} C_VEL
LIN {X 0,Y 144.498,Z 439.904,A -85,B 0,C 180,E1 -25783.153,E2 -25783.153} C_VEL
LIN {X 0,Y 137.241,Z 448.423,A -85,B 0,C 180,E1 -25787.274,E2 -25787.274} C_VEL
LIN {X 0,Y 130.701,Z 455.512,A -85,B 0,C 180,E1 -25791.805,E2 -25791.805} C_VEL
LIN {X 0,Y 124.316,Z 462.088,A -85,B 0,C 180,E1 -25797.518,E2 -25797.518} C_VEL
LIN {X 0,Y 119.246,Z 467.226,A -85,B 0,C 180,E1 -25803.769,E2 -25803.769} C_VEL
LIN {X 0,Y 116.27,Z 470.187,A -85,B 0,C 180,E1 -25808.737,E2 -25808.737} C_VEL
LIN {X 0,Y 113.661,Z 473.079,A -85,B 0,C 180,E1 -25815.682,E2 -25815.682} C_VEL
LIN {X 0,Y 112.348,Z 474.813,A -85,B 0,C 180,E1 -25822.814,E2 -25822.814} C_VEL
LIN {X 0,Y 112.199,Z 475.413,A -85,B 0,C 180,E1 -25830.001,E2 -25830.001} C_VEL
LIN {X 0,Y 112.347,Z 474.843,A -85,B 0,C 180,E1 -25837.189,E2 -25837.189} C_VEL
LIN {X 0,Y 113.636,Z 473.15,A -85,B 0,C 180,E1 -25844.324,E2 -25844.324} C_VEL
LIN {X 0,Y 116.237,Z 470.293,A -85,B 0,C 180,E1 -25851.272,E2 -25851.272} C_VEL
LIN {X 0,Y 120.324,Z 466.204,A -85,B 0,C 180,E1 -25857.858,E2 -25857.858} C_VEL
LIN {X 0,Y 125.727,Z 460.784,A -85,B 0,C 180,E1 -25863.987,E2 -25863.987} C_VEL
LIN {X 0,Y 132.409,Z 453.877,A -85,B 0,C 180,E1 -25869.564,E2 -25869.564} C_VEL
LIN {X 0,Y 139.225,Z 446.457,A -85,B 0,C 180,E1 -25873.956,E2 -25873.956} C_VEL
LIN {X 0,Y 146.336,Z 437.784,A -85,B 0,C 180,E1 -25877.903,E2 -25877.903} C_VEL
LIN {X 0,Y 153.476,Z 428.392,A -85,B 0,C 180,E1 -25881.121,E2 -25881.121} C_VEL
LIN {X 0,Y 159.085,Z 420.264,A -85,B 0,C 180,E1 -25883.358,E2 -25883.358} C_VEL
LIN {X 0,Y 160.679,Z 413.663,A -85,B 0,C 180,E1 -25886.207,E2 -25886.207} C_VEL
LIN {X 0,Y 161.392,Z 408.737,A -85,B 0,C 180,E1 -25888.496,E2 -25888.496} C_VEL
LIN {X 0,Y 161.283,Z 403.539,A -85,B 0,C 180,E1 -25891.358,E2 -25891.358} C_VEL
LIN {X 0,Y 160.635,Z 397.032,A -85,B 0,C 180,E1 -25895.44,E2 -25895.44} C_VEL
LIN {X 0,Y 159.706,Z 391.728,A -85,B 0,C 180,E1 -25899.387,E2 -25899.387} C_VEL
LIN {X 0,Y 158.607,Z 387.729,A -85,B 0,C 180,E1 -25903.26,E2 -25903.26} C_VEL
LIN {X 0,Y 157.556,Z 384.763,A -85,B 0,C 180,E1 -25907.113,E2 -25907.113} C_VEL
LIN {X 0,Y 157.012,Z 382.966,A -85,B 0,C 180,E1 -25909.979,E2 -25909.979} C_VEL
LIN {X 0,Y 156.123,Z 381.343,A -85,B 0,C 180,E1 -25914.834,E2 -25914.834} C_VEL
LIN {X 0,Y 156.191,Z 380.057,A -85,B 0,C 180,E1 -25920,E2 -25920} C_VEL
LIN {X 0,Y 156.693,Z 382.101,A -85,B 0,C 180,E1 -25927.733,E2 -25927.733} C_VEL
LIN {X 0,Y 157.265,Z 383.469,A -85,B 0,C 180,E1 -25930.531,E2 -25930.531} C_VEL
LIN {X 0,Y 158.066,Z 386.003,A -85,B 0,C 180,E1 -25934.155,E2 -25934.155} C_VEL
LIN {X 0,Y 158.966,Z 389.886,A -85,B 0,C 180,E1 -25938.027,E2 -25938.027} C_VEL
LIN {X 0,Y 160.017,Z 395.872,A -85,B 0,C 180,E1 -25942.731,E2 -25942.731} C_VEL
LIN {X 0,Y 160.721,Z 402.03,A -85,B 0,C 180,E1 -25946.715,E2 -25946.715} C_VEL
LIN {X 0,Y 161.039,Z 408.005,A -85,B 0,C 180,E1 -25950.123,E2 -25950.123} C_VEL
LIN {X 0,Y 160.557,Z 412.6,A -85,B 0,C 180,E1 -25952.284,E2 -25952.284} C_VEL
LIN {X 0,Y 158.59,Z 421.076,A -85,B 0,C 180,E1 -25955.887,E2 -25955.887} C_VEL
LIN {X 0,Y 157.888,Z 423.233,A -85,B 0,C 180,E1 -25956.752,E2 -25956.752} C_VEL
LIN {X 0,Y 150.668,Z 433.445,A -85,B 0,C 180,E1 -25959.677,E2 -25959.677} C_VEL
LIN {X 0,Y 142.747,Z 443.417,A -85,B 0,C 180,E1 -25963.429,E2 -25963.429} C_VEL
LIN {X 0,Y 135.718,Z 451.706,A -85,B 0,C 180,E1 -25967.686,E2 -25967.686} C_VEL
LIN {X 0,Y 130.099,Z 457.674,A -85,B 0,C 180,E1 -25971.593,E2 -25971.593} C_VEL
LIN {X 0,Y 123.706,Z 464.249,A -85,B 0,C 180,E1 -25977.335,E2 -25977.335} C_VEL
LIN {X 0,Y 118.739,Z 469.395,A -85,B 0,C 180,E1 -25983.645,E2 -25983.645} C_VEL
LIN {X 0,Y 115.891,Z 472.374,A -85,B 0,C 180,E1 -25988.662,E2 -25988.662} C_VEL
LIN {X 0,Y 113.334,Z 475.274,A -85,B 0,C 180,E1 -25995.637,E2 -25995.637} C_VEL
LIN {X 0,Y 112.218,Z 477.004,A -85,B 0,C 180,E1 -26002.803,E2 -26002.803} C_VEL
LIN {X 0,Y 112.133,Z 477.595,A -85,B 0,C 180,E1 -26009.999,E2 -26009.999} C_VEL
LIN {X 0,Y 112.217,Z 476.985,A -85,B 0,C 180,E1 -26017.194,E2 -26017.194} C_VEL
LIN {X 0,Y 113.333,Z 475.231,A -85,B 0,C 180,E1 -26024.36,E2 -26024.36} C_VEL
LIN {X 0,Y 115.892,Z 472.312,A -85,B 0,C 180,E1 -26031.335,E2 -26031.335} C_VEL
LIN {X 0,Y 119.844,Z 468.157,A -85,B 0,C 180,E1 -26037.977,E2 -26037.977} C_VEL
LIN {X 0,Y 125.197,Z 462.657,A -85,B 0,C 180,E1 -26044.147,E2 -26044.147} C_VEL
LIN {X 0,Y 131.855,Z 455.663,A -85,B 0,C 180,E1 -26049.761,E2 -26049.761} C_VEL
LIN {X 0,Y 138.673,Z 448.185,A -85,B 0,C 180,E1 -26054.173,E2 -26054.173} C_VEL
LIN {X 0,Y 146.069,Z 439.165,A -85,B 0,C 180,E1 -26058.222,E2 -26058.222} C_VEL
LIN {X 0,Y 154.21,Z 428.322,A -85,B 0,C 180,E1 -26061.825,E2 -26061.825} C_VEL
LIN {X 0,Y 157.844,Z 422.981,A -85,B 0,C 180,E1 -26063.266,E2 -26063.266} C_VEL
LIN {X 0,Y 159.85,Z 415.487,A -85,B 0,C 180,E1 -26066.393,E2 -26066.393} C_VEL
LIN {X 0,Y 160.691,Z 411.006,A -85,B 0,C 180,E1 -26068.343,E2 -26068.343} C_VEL
LIN {X 0,Y 160.922,Z 407.843,A -85,B 0,C 180,E1 -26069.853,E2 -26069.853} C_VEL
LIN {X 0,Y 160.576,Z 401.624,A -85,B 0,C 180,E1 -26073.395,E2 -26073.395} C_VEL
LIN {X 0,Y 159.86,Z 395.679,A -85,B 0,C 180,E1 -26077.257,E2 -26077.257} C_VEL
LIN {X 0,Y 159.434,Z 392.761,A -85,B 0,C 180,E1 -26079.351,E2 -26079.351} C_VEL
LIN {X 0,Y 158.458,Z 388.302,A -85,B 0,C 180,E1 -26083.245,E2 -26083.245} C_VEL
LIN {X 0,Y 157.606,Z 384.755,A -85,B 0,C 180,E1 -26087.117,E2 -26087.117} C_VEL
LIN {X 0,Y 157.534,Z 384.575,A -85,B 0,C 180,E1 -26087.387,E2 -26087.387} C_VEL
LIN {X 0,Y 156.687,Z 383.923,A -85,B 0,C 180,E1 -26089.5,E2 -26089.5} C_VEL
LIN {X 0,Y 155.455,Z 384.334,A -85,B 0,C 180,E1 -26091.632,E2 -26091.632} C_VEL
LIN {X 0,Y 153.119,Z 386.121,A -85,B 0,C 180,E1 -26095.973,E2 -26095.973} C_VEL
LIN {X 0,Y 152.631,Z 386.388,A -85,B 0,C 180,E1 -26098.212,E2 -26098.212} C_VEL
LIN {X 0,Y 152.652,Z 386.241,A -85,B 0,C 180,E1 -26098.96,E2 -26098.96} C_VEL
LIN {X 0,Y 152.781,Z 385.933,A -85,B 0,C 180,E1 -26100,E2 -26100} C_VEL
LIN {X 0,Y 152.944,Z 388.051,A -85,B 0,C 180,E1 -26107.924,E2 -26107.924} C_VEL
LIN {X 0,Y 153.394,Z 389.216,A -85,B 0,C 180,E1 -26110.56,E2 -26110.56} C_VEL
LIN {X 0,Y 154.382,Z 392.847,A -85,B 0,C 180,E1 -26115.852,E2 -26115.852} C_VEL
LIN {X 0,Y 155.321,Z 396.618,A -85,B 0,C 180,E1 -26119.838,E2 -26119.838} C_VEL
LIN {X 0,Y 155.881,Z 401.853,A -85,B 0,C 180,E1 -26123.94,E2 -26123.94} C_VEL
LIN {X 0,Y 156.127,Z 407.134,A -85,B 0,C 180,E1 -26127.478,E2 -26127.478} C_VEL
LIN {X 0,Y 156.016,Z 412.018,A -85,B 0,C 180,E1 -26130.39,E2 -26130.39} C_VEL
LIN {X 0,Y 154.886,Z 417.866,A -85,B 0,C 180,E1 -26133.272,E2 -26133.272} C_VEL
LIN {X 0,Y 153.993,Z 421.136,A -85,B 0,C 180,E1 -26134.769,E2 -26134.769} C_VEL
LIN {X 0,Y 151.7,Z 424.69,A -85,B 0,C 180,E1 -26135.834,E2 -26135.834} C_VEL
LIN {X 0,Y 144.33,Z 434.348,A -85,B 0,C 180,E1 -26138.824,E2 -26138.824} C_VEL
LIN {X 0,Y 136.426,Z 443.816,A -85,B 0,C 180,E1 -26142.772,E2 -26142.772} C_VEL
LIN {X 0,Y 128.97,Z 451.701,A -85,B 0,C 180,E1 -26147.068,E2 -26147.068} C_VEL
LIN {X 0,Y 121.592,Z 459.061,A -85,B 0,C 180,E1 -26152.637,E2 -26152.637} C_VEL
LIN {X 0,Y 116.196,Z 464.157,A -85,B 0,C 180,E1 -26157.863,E2 -26157.863} C_VEL
LIN {X 0,Y 111.76,Z 468.355,A -85,B 0,C 180,E1 -26163.886,E2 -26163.886} C_VEL
LIN {X 0,Y 107.99,Z 471.852,A -85,B 0,C 180,E1 -26171.012,E2 -26171.012} C_VEL
LIN {X 0,Y 105.844,Z 474.157,A -85,B 0,C 180,E1 -26178.512,E2 -26178.512} C_VEL
LIN {X 0,Y 105.045,Z 475.327,A -85,B 0,C 180,E1 -26186.165,E2 -26186.165} C_VEL
LIN {X 0,Y 105.106,Z 475.482,A -85,B 0,C 180,E1 -26190.001,E2 -26190.001} C_VEL
LIN {X 0,Y 105.29,Z 474.912,A -85,B 0,C 180,E1 -26197.673,E2 -26197.673} C_VEL
LIN {X 0,Y 106.734,Z 473.219,A -85,B 0,C 180,E1 -26205.272,E2 -26205.272} C_VEL
LIN {X 0,Y 109.624,Z 470.362,A -85,B 0,C 180,E1 -26212.624,E2 -26212.624} C_VEL
LIN {X 0,Y 114.05,Z 466.272,A -85,B 0,C 180,E1 -26219.537,E2 -26219.537} C_VEL
LIN {X 0,Y 119.865,Z 460.852,A -85,B 0,C 180,E1 -26225.898,E2 -26225.898} C_VEL
LIN {X 0,Y 126.976,Z 453.945,A -85,B 0,C 180,E1 -26231.621,E2 -26231.621} C_VEL
LIN {X 0,Y 134.169,Z 446.525,A -85,B 0,C 180,E1 -26236.076,E2 -26236.076} C_VEL
LIN {X 0,Y 141.877,Z 437.584,A -85,B 0,C 180,E1 -26240.156,E2 -26240.156} C_VEL
LIN {X 0,Y 149.098,Z 428.458,A -85,B 0,C 180,E1 -26243.257,E2 -26243.257} C_VEL
LIN {X 0,Y 154.029,Z 421.532,A -85,B 0,C 180,E1 -26245.215,E2 -26245.215} C_VEL
LIN {X 0,Y 155.585,Z 415.578,A -85,B 0,C 180,E1 -26248.018,E2 -26248.018} C_VEL
LIN {X 0,Y 156.221,Z 411.074,A -85,B 0,C 180,E1 -26250.339,E2 -26250.339} C_VEL
LIN {X 0,Y 156.203,Z 404.94,A -85,B 0,C 180,E1 -26254.14,E2 -26254.14} C_VEL
LIN {X 0,Y 155.759,Z 399.567,A -85,B 0,C 180,E1 -26258.011,E2 -26258.011} C_VEL
LIN {X 0,Y 155.15,Z 395.584,A -85,B 0,C 180,E1 -26261.513,E2 -26261.513} C_VEL
LIN {X 0,Y 154.574,Z 393.106,A -85,B 0,C 180,E1 -26264.169,E2 -26264.169} C_VEL
LIN {X 0,Y 153.541,Z 389.577,A -85,B 0,C 180,E1 -26269.45,E2 -26269.45} C_VEL
LIN {X 0,Y 153.129,Z 388.339,A -85,B 0,C 180,E1 -26272.086,E2 -26272.086} C_VEL
LIN {X 0,Y 152.88,Z 386.352,A -85,B 0,C 180,E1 -26280,E2 -26280} C_VEL
LIN {X 0,Y 153.28,Z 388.443,A -85,B 0,C 180,E1 -26287.906,E2 -26287.906} C_VEL
LIN {X 0,Y 153.719,Z 389.76,A -85,B 0,C 180,E1 -26290.537,E2 -26290.537} C_VEL
LIN {X 0,Y 154.363,Z 392.651,A -85,B 0,C 180,E1 -26294.501,E2 -26294.501} C_VEL
LIN {X 0,Y 155.032,Z 396.68,A -85,B 0,C 180,E1 -26298.501,E2 -26298.501} C_VEL
LIN {X 0,Y 155.576,Z 401.798,A -85,B 0,C 180,E1 -26302.585,E2 -26302.585} C_VEL
LIN {X 0,Y 155.88,Z 408.114,A -85,B 0,C 180,E1 -26306.799,E2 -26306.799} C_VEL
LIN {X 0,Y 155.832,Z 412.204,A -85,B 0,C 180,E1 -26309.231,E2 -26309.231} C_VEL
LIN {X 0,Y 155.092,Z 416.64,A -85,B 0,C 180,E1 -26311.406,E2 -26311.406} C_VEL
LIN {X 0,Y 153.217,Z 423.158,A -85,B 0,C 180,E1 -26314.345,E2 -26314.345} C_VEL
LIN {X 0,Y 152.453,Z 424.951,A -85,B 0,C 180,E1 -26315.088,E2 -26315.088} C_VEL
LIN {X 0,Y 144.978,Z 434.884,A -85,B 0,C 180,E1 -26318.025,E2 -26318.025} C_VEL
LIN {X 0,Y 137.201,Z 444.158,A -85,B 0,C 180,E1 -26321.637,E2 -26321.637} C_VEL
LIN {X 0,Y 129.499,Z 452.712,A -85,B 0,C 180,E1 -26326.215,E2 -26326.215} C_VEL
LIN {X 0,Y 122.763,Z 459.419,A -85,B 0,C 180,E1 -26330.969,E2 -26330.969} C_VEL
LIN {X 0,Y 116.243,Z 465.608,A -85,B 0,C 180,E1 -26337.033,E2 -26337.033} C_VEL
LIN {X 0,Y 111.222,Z 470.397,A -85,B 0,C 180,E1 -26343.747,E2 -26343.747} C_VEL
LIN {X 0,Y 107.599,Z 473.905,A -85,B 0,C 180,E1 -26350.937,E2 -26350.937} C_VEL
LIN {X 0,Y 105.605,Z 476.213,A -85,B 0,C 180,E1 -26358.482,E2 -26358.482} C_VEL
LIN {X 0,Y 104.958,Z 477.373,A -85,B 0,C 180,E1 -26366.159,E2 -26366.159} C_VEL
LIN {X 0,Y 105.033,Z 477.526,A -85,B 0,C 180,E1 -26369.999,E2 -26369.999} C_VEL
LIN {X 0,Y 105.154,Z 476.916,A -85,B 0,C 180,E1 -26377.68,E2 -26377.68} C_VEL
LIN {X 0,Y 106.426,Z 475.161,A -85,B 0,C 180,E1 -26385.314,E2 -26385.314} C_VEL
LIN {X 0,Y 109.254,Z 472.241,A -85,B 0,C 180,E1 -26392.702,E2 -26392.702} C_VEL
LIN {X 0,Y 114.151,Z 467.499,A -85,B 0,C 180,E1 -26400.465,E2 -26400.465} C_VEL
LIN {X 0,Y 119.326,Z 462.586,A -85,B 0,C 180,E1 -26406.082,E2 -26406.082} C_VEL
LIN {X 0,Y 126.447,Z 455.592,A -85,B 0,C 180,E1 -26411.831,E2 -26411.831} C_VEL
LIN {X 0,Y 133.603,Z 448.113,A -85,B 0,C 180,E1 -26416.325,E2 -26416.325} C_VEL
LIN {X 0,Y 141.41,Z 439.094,A -85,B 0,C 180,E1 -26420.382,E2 -26420.382} C_VEL
LIN {X 0,Y 149.899,Z 428.25,A -85,B 0,C 180,E1 -26423.972,E2 -26423.972} C_VEL
LIN {X 0,Y 152.445,Z 424.694,A -85,B 0,C 180,E1 -26424.913,E2 -26424.913} C_VEL
LIN {X 0,Y 154.348,Z 418.773,A -85,B 0,C 180,E1 -26427.527,E2 -26427.527} C_VEL
LIN {X 0,Y 155.623,Z 413.023,A -85,B 0,C 180,E1 -26430.214,E2 -26430.214} C_VEL
LIN {X 0,Y 155.773,Z 407.919,A -85,B 0,C 180,E1 -26433.182,E2 -26433.182} C_VEL
LIN {X 0,Y 155.549,Z 402.423,A -85,B 0,C 180,E1 -26436.786,E2 -26436.786} C_VEL
LIN {X 0,Y 155.146,Z 397.979,A -85,B 0,C 180,E1 -26440.139,E2 -26440.139} C_VEL
LIN {X 0,Y 154.427,Z 393.644,A -85,B 0,C 180,E1 -26444.154,E2 -26444.154} C_VEL
LIN {X 0,Y 154.053,Z 391.243,A -85,B 0,C 180,E1 -26446.815,E2 -26446.815} C_VEL
LIN {X 0,Y 153.562,Z 389.494,A -85,B 0,C 180,E1 -26449.452,E2 -26449.452} C_VEL
LIN {X 0,Y 153.094,Z 388.217,A -85,B 0,C 180,E1 -26452.084,E2 -26452.084} C_VEL
LIN {X 0,Y 152.652,Z 386.241,A -85,B 0,C 180,E1 -26458.96,E2 -26458.96} C_VEL
LIN {X 0,Y 152.613,Z 386.249,A -85,B 0,C 180,E1 -26460.42,E2 -26460.42} C_VEL
LIN {X 0,Y 152.05,Z 387.506,A -85,B 0,C 180,E1 -26462.573,E2 -26462.573} C_VEL
LIN {X 0,Y 150.476,Z 391.301,A -85,B 0,C 180,E1 -26466.05,E2 -26466.05} C_VEL
LIN {X 0,Y 149.544,Z 394.319,A -85,B 0,C 180,E1 -26468.93,E2 -26468.93} C_VEL
LIN {X 0,Y 149.566,Z 395.311,A -85,B 0,C 180,E1 -26470.44,E2 -26470.44} C_VEL
LIN {X 0,Y 150.212,Z 398.163,A -85,B 0,C 180,E1 -26474.912,E2 -26474.912} C_VEL
LIN {X 0,Y 150.89,Z 401.741,A -85,B 0,C 180,E1 -26479.029,E2 -26479.029} C_VEL
LIN {X 0,Y 151.127,Z 406.853,A -85,B 0,C 180,E1 -26483.284,E2 -26483.284} C_VEL
LIN {X 0,Y 151.065,Z 411.638,A -85,B 0,C 180,E1 -26486.675,E2 -26486.675} C_VEL
LIN {X 0,Y 150.772,Z 415.777,A -85,B 0,C 180,E1 -26489.303,E2 -26489.303} C_VEL
LIN {X 0,Y 149.378,Z 421.221,A -85,B 0,C 180,E1 -26492.13,E2 -26492.13} C_VEL
LIN {X 0,Y 148.766,Z 422.987,A -85,B 0,C 180,E1 -26493.016,E2 -26493.016} C_VEL
LIN {X 0,Y 146.342,Z 426.531,A -85,B 0,C 180,E1 -26494.066,E2 -26494.066} C_VEL
LIN {X 0,Y 138.62,Z 436.05,A -85,B 0,C 180,E1 -26497.135,E2 -26497.135} C_VEL
LIN {X 0,Y 130.545,Z 445.115,A -85,B 0,C 180,E1 -26501.091,E2 -26501.091} C_VEL
LIN {X 0,Y 122.803,Z 452.777,A -85,B 0,C 180,E1 -26505.49,E2 -26505.49} C_VEL
LIN {X 0,Y 116,Z 459.132,A -85,B 0,C 180,E1 -26510.497,E2 -26510.497} C_VEL
LIN {X 0,Y 109.801,Z 464.56,A -85,B 0,C 180,E1 -26516.315,E2 -26516.315} C_VEL
LIN {X 0,Y 105.378,Z 468.425,A -85,B 0,C 180,E1 -26522.172,E2 -26522.172} C_VEL
LIN {X 0,Y 101.255,Z 471.922,A -85,B 0,C 180,E1 -26529.695,E2 -26529.695} C_VEL
LIN {X 0,Y 98.887,Z 474.227,A -85,B 0,C 180,E1 -26537.691,E2 -26537.691} C_VEL
LIN {X 0,Y 97.952,Z 475.397,A -85,B 0,C 180,E1 -26545.887,E2 -26545.887} C_VEL
LIN {X 0,Y 98.006,Z 475.551,A -85,B 0,C 180,E1 -26550.002,E2 -26550.002} C_VEL
LIN {X 0,Y 98.257,Z 474.981,A -85,B 0,C 180,E1 -26558.226,E2 -26558.226} C_VEL
LIN {X 0,Y 99.852,Z 473.288,A -85,B 0,C 180,E1 -26566.353,E2 -26566.353} C_VEL
LIN {X 0,Y 103.08,Z 470.43,A -85,B 0,C 180,E1 -26574.148,E2 -26574.148} C_VEL
LIN {X 0,Y 107.885,Z 466.341,A -85,B 0,C 180,E1 -26581.41,E2 -26581.41} C_VEL
LIN {X 0,Y 114.148,Z 460.92,A -85,B 0,C 180,E1 -26588.003,E2 -26588.003} C_VEL
LIN {X 0,Y 121.705,Z 454.013,A -85,B 0,C 180,E1 -26593.865,E2 -26593.865} C_VEL
LIN {X 0,Y 130.455,Z 445.392,A -85,B 0,C 180,E1 -26598.958,E2 -26598.958} C_VEL
LIN {X 0,Y 137.426,Z 437.648,A -85,B 0,C 180,E1 -26602.437,E2 -26602.437} C_VEL
LIN {X 0,Y 144.95,Z 428.525,A -85,B 0,C 180,E1 -26605.514,E2 -26605.514} C_VEL
LIN {X 0,Y 148.78,Z 423.378,A -85,B 0,C 180,E1 -26606.979,E2 -26606.979} C_VEL
LIN {X 0,Y 150.482,Z 417.671,A -85,B 0,C 180,E1 -26609.864,E2 -26609.864} C_VEL
LIN {X 0,Y 151.027,Z 414.786,A -85,B 0,C 180,E1 -26611.513,E2 -26611.513} C_VEL
LIN {X 0,Y 151.304,Z 409.13,A -85,B 0,C 180,E1 -26615.288,E2 -26615.288} C_VEL
LIN {X 0,Y 151.192,Z 405.055,A -85,B 0,C 180,E1 -26618.385,E2 -26618.385} C_VEL
LIN {X 0,Y 151.015,Z 402.077,A -85,B 0,C 180,E1 -26620.987,E2 -26620.987} C_VEL
LIN {X 0,Y 150.379,Z 398.428,A -85,B 0,C 180,E1 -26625.105,E2 -26625.105} C_VEL
LIN {X 0,Y 149.566,Z 395.09,A -85,B 0,C 180,E1 -26630.673,E2 -26630.673} C_VEL
LIN {X 0,Y 149.131,Z 393.757,A -85,B 0,C 180,E1 -26634.591,E2 -26634.591} C_VEL
LIN {X 0,Y 149.315,Z 392.509,A -85,B 0,C 180,E1 -26640,E2 -26640} C_VEL
LIN {X 0,Y 149.596,Z 394.667,A -85,B 0,C 180,E1 -26648.102,E2 -26648.102} C_VEL
LIN {X 0,Y 149.949,Z 396.048,A -85,B 0,C 180,E1 -26650.805,E2 -26650.805} C_VEL
LIN {X 0,Y 150.39,Z 399.119,A -85,B 0,C 180,E1 -26654.893,E2 -26654.893} C_VEL
LIN {X 0,Y 150.788,Z 403.328,A -85,B 0,C 180,E1 -26659.042,E2 -26659.042} C_VEL
LIN {X 0,Y 150.916,Z 408.749,A -85,B 0,C 180,E1 -26663.318,E2 -26663.318} C_VEL
LIN {X 0,Y 150.669,Z 415.454,A -85,B 0,C 180,E1 -26667.804,E2 -26667.804} C_VEL
LIN {X 0,Y 149.744,Z 419.707,A -85,B 0,C 180,E1 -26670.087,E2 -26670.087} C_VEL
LIN {X 0,Y 147.838,Z 425.368,A -85,B 0,C 180,E1 -26672.8,E2 -26672.8} C_VEL
LIN {X 0,Y 147.146,Z 426.669,A -85,B 0,C 180,E1 -26673.297,E2 -26673.297} C_VEL
LIN {X 0,Y 139.432,Z 436.304,A -85,B 0,C 180,E1 -26676.247,E2 -26676.247} C_VEL
LIN {X 0,Y 131.039,Z 445.667,A -85,B 0,C 180,E1 -26680.06,E2 -26680.06} C_VEL
LIN {X 0,Y 123.377,Z 453.655,A -85,B 0,C 180,E1 -26684.598,E2 -26684.598} C_VEL
LIN {X 0,Y 115.42,Z 461.014,A -85,B 0,C 180,E1 -26690.255,E2 -26690.255} C_VEL
LIN {X 0,Y 108.63,Z 466.978,A -85,B 0,C 180,E1 -26696.859,E2 -26696.859} C_VEL
LIN {X 0,Y 104.851,Z 470.328,A -85,B 0,C 180,E1 -26702.017,E2 -26702.017} C_VEL
LIN {X 0,Y 100.861,Z 473.836,A -85,B 0,C 180,E1 -26709.609,E2 -26709.609} C_VEL
LIN {X 0,Y 98.632,Z 476.144,A -85,B 0,C 180,E1 -26717.656,E2 -26717.656} C_VEL
LIN {X 0,Y 97.883,Z 477.304,A -85,B 0,C 180,E1 -26725.881,E2 -26725.881} C_VEL
LIN {X 0,Y 97.94,Z 477.457,A -85,B 0,C 180,E1 -26729.998,E2 -26729.998} C_VEL
LIN {X 0,Y 98.094,Z 476.846,A -85,B 0,C 180,E1 -26738.237,E2 -26738.237} C_VEL
LIN {X 0,Y 99.561,Z 475.091,A -85,B 0,C 180,E1 -26746.399,E2 -26746.399} C_VEL
LIN {X 0,Y 102.691,Z 472.171,A -85,B 0,C 180,E1 -26754.242,E2 -26754.242} C_VEL
LIN {X 0,Y 107.691,Z 467.736,A -85,B 0,C 180,E1 -26761.964,E2 -26761.964} C_VEL
LIN {X 0,Y 113.62,Z 462.515,A -85,B 0,C 180,E1 -26768.208,E2 -26768.208} C_VEL
LIN {X 0,Y 121.228,Z 455.522,A -85,B 0,C 180,E1 -26774.079,E2 -26774.079} C_VEL
LIN {X 0,Y 127.667,Z 449.165,A -85,B 0,C 180,E1 -26777.999,E2 -26777.999} C_VEL
LIN {X 0,Y 135.752,Z 440.378,A -85,B 0,C 180,E1 -26782.136,E2 -26782.136} C_VEL
LIN {X 0,Y 144.509,Z 429.814,A -85,B 0,C 180,E1 -26785.766,E2 -26785.766} C_VEL
LIN {X 0,Y 147.14,Z 426.406,A -85,B 0,C 180,E1 -26786.704,E2 -26786.704} C_VEL
LIN {X 0,Y 148.847,Z 422.067,A -85,B 0,C 180,E1 -26788.71,E2 -26788.71} C_VEL
LIN {X 0,Y 150.379,Z 416.676,A -85,B 0,C 180,E1 -26791.378,E2 -26791.378} C_VEL
LIN {X 0,Y 150.756,Z 411.589,A -85,B 0,C 180,E1 -26794.56,E2 -26794.56} C_VEL
LIN {X 0,Y 150.745,Z 405.705,A -85,B 0,C 180,E1 -26798.812,E2 -26798.812} C_VEL
LIN {X 0,Y 150.541,Z 401.929,A -85,B 0,C 180,E1 -26802.018,E2 -26802.018} C_VEL
LIN {X 0,Y 150.191,Z 397.645,A -85,B 0,C 180,E1 -26806.469,E2 -26806.469} C_VEL
LIN {X 0,Y 149.618,Z 395.046,A -85,B 0,C 180,E1 -26810.539,E2 -26810.539} C_VEL
LIN {X 0,Y 149.088,Z 393.571,A -85,B 0,C 180,E1 -26814.59,E2 -26814.59} C_VEL
LIN {X 0,Y 149.219,Z 392.135,A -85,B 0,C 180,E1 -26820,E2 -26820} C_VEL
LIN {X 0,Y 149.352,Z 394.553,A -85,B 0,C 180,E1 -26828.828,E2 -26828.828} C_VEL
LIN {X 0,Y 149.566,Z 395.311,A -85,B 0,C 180,E1 -26830.44,E2 -26830.44} C_VEL
LIN {X 0,Y 149.65,Z 396.329,A -85,B 0,C 180,E1 -26831.894,E2 -26831.894} C_VEL
LIN {X 0,Y 149.399,Z 397.856,A -85,B 0,C 180,E1 -26833.283,E2 -26833.283} C_VEL
LIN {X 0,Y 148.333,Z 401.818,A -85,B 0,C 180,E1 -26835.907,E2 -26835.907} C_VEL
LIN {X 0,Y 146.522,Z 408.322,A -85,B 0,C 180,E1 -26839.875,E2 -26839.875} C_VEL
LIN {X 0,Y 146.329,Z 410.141,A -85,B 0,C 180,E1 -26841.295,E2 -26841.295} C_VEL
LIN {X 0,Y 146.103,Z 414.611,A -85,B 0,C 180,E1 -26844.832,E2 -26844.832} C_VEL
LIN {X 0,Y 145.539,Z 418.954,A -85,B 0,C 180,E1 -26847.859,E2 -26847.859} C_VEL
LIN {X 0,Y 144.363,Z 423.021,A -85,B 0,C 180,E1 -26850.181,E2 -26850.181} C_VEL
LIN {X 0,Y 143.678,Z 424.837,A -85,B 0,C 180,E1 -26851.132,E2 -26851.132} C_VEL
LIN {X 0,Y 141.122,Z 428.236,A -85,B 0,C 180,E1 -26852.158,E2 -26852.158} C_VEL
LIN {X 0,Y 133.04,Z 437.69,A -85,B 0,C 180,E1 -26855.3,E2 -26855.3} C_VEL
LIN {X 0,Y 124.768,Z 446.404,A -85,B 0,C 180,E1 -26859.242,E2 -26859.242} C_VEL
LIN {X 0,Y 116.716,Z 453.853,A -85,B 0,C 180,E1 -26863.736,E2 -26863.736} C_VEL
LIN {X 0,Y 108.674,Z 460.81,A -85,B 0,C 180,E1 -26869.709,E2 -26869.709} C_VEL
LIN {X 0,Y 101.91,Z 466.275,A -85,B 0,C 180,E1 -26876.518,E2 -26876.518} C_VEL
LIN {X 0,Y 96.655,Z 470.397,A -85,B 0,C 180,E1 -26884.136,E2 -26884.136} C_VEL
LIN {X 0,Y 93.054,Z 473.289,A -85,B 0,C 180,E1 -26892.418,E2 -26892.418} C_VEL
LIN {X 0,Y 91.225,Z 475.021,A -85,B 0,C 180,E1 -26901.138,E2 -26901.138} C_VEL
LIN {X 0,Y 90.913,Z 475.62,A -85,B 0,C 180,E1 -26910.002,E2 -26910.002} C_VEL
LIN {X 0,Y 91.224,Z 475.05,A -85,B 0,C 180,E1 -26918.865,E2 -26918.865} C_VEL
LIN {X 0,Y 93.017,Z 473.357,A -85,B 0,C 180,E1 -26927.593,E2 -26927.593} C_VEL
LIN {X 0,Y 96.62,Z 470.499,A -85,B 0,C 180,E1 -26935.878,E2 -26935.878} C_VEL
LIN {X 0,Y 101.834,Z 466.41,A -85,B 0,C 180,E1 -26943.513,E2 -26943.513} C_VEL
LIN {X 0,Y 108.597,Z 460.988,A -85,B 0,C 180,E1 -26950.329,E2 -26950.329} C_VEL
LIN {X 0,Y 116.643,Z 454.081,A -85,B 0,C 180,E1 -26956.306,E2 -26956.306} C_VEL
LIN {X 0,Y 124.692,Z 446.66,A -85,B 0,C 180,E1 -26960.805,E2 -26960.805} C_VEL
LIN {X 0,Y 131.93,Z 439.066,A -85,B 0,C 180,E1 -26964.329,E2 -26964.329} C_VEL
LIN {X 0,Y 141.044,Z 428.591,A -85,B 0,C 180,E1 -26967.897,E2 -26967.897} C_VEL
LIN {X 0,Y 143.686,Z 425.223,A -85,B 0,C 180,E1 -26968.867,E2 -26968.867} C_VEL
LIN {X 0,Y 145.599,Z 419.403,A -85,B 0,C 180,E1 -26972.075,E2 -26972.075} C_VEL
LIN {X 0,Y 146.268,Z 413.938,A -85,B 0,C 180,E1 -26975.913,E2 -26975.913} C_VEL
LIN {X 0,Y 146.463,Z 409.609,A -85,B 0,C 180,E1 -26979.46,E2 -26979.46} C_VEL
LIN {X 0,Y 146.436,Z 407.059,A -85,B 0,C 180,E1 -26981.822,E2 -26981.822} C_VEL
LIN {X 0,Y 146.057,Z 403.633,A -85,B 0,C 180,E1 -26986.078,E2 -26986.078} C_VEL
LIN {X 0,Y 145.506,Z 400.581,A -85,B 0,C 180,E1 -26991.668,E2 -26991.668} C_VEL
LIN {X 0,Y 145.499,Z 398.528,A -85,B 0,C 180,E1 -27000,E2 -27000} C_VEL
LIN {X 0,Y 145.672,Z 400.72,A -85,B 0,C 180,E1 -27008.322,E2 -27008.322} C_VEL
LIN {X 0,Y 146.015,Z 403.15,A -85,B 0,C 180,E1 -27012.509,E2 -27012.509} C_VEL
LIN {X 0,Y 146.144,Z 406.799,A -85,B 0,C 180,E1 -27016.77,E2 -27016.77} C_VEL
LIN {X 0,Y 146.093,Z 411.663,A -85,B 0,C 180,E1 -27021.146,E2 -27021.146} C_VEL
LIN {X 0,Y 145.736,Z 416.465,A -85,B 0,C 180,E1 -27024.738,E2 -27024.738} C_VEL
LIN {X 0,Y 145.069,Z 420.77,A -85,B 0,C 180,E1 -27027.612,E2 -27027.612} C_VEL
LIN {X 0,Y 143.357,Z 425.56,A -85,B 0,C 180,E1 -27030.118,E2 -27030.118} C_VEL
LIN {X 0,Y 142.751,Z 427.086,A -85,B 0,C 180,E1 -27030.884,E2 -27030.884} C_VEL
LIN {X 0,Y 141.814,Z 428.581,A -85,B 0,C 180,E1 -27031.44,E2 -27031.44} C_VEL
LIN {X 0,Y 132.736,Z 439.152,A -85,B 0,C 180,E1 -27034.846,E2 -27034.846} C_VEL
LIN {X 0,Y 124.089,Z 448.144,A -85,B 0,C 180,E1 -27038.852,E2 -27038.852} C_VEL
LIN {X 0,Y 116.222,Z 455.606,A -85,B 0,C 180,E1 -27043.476,E2 -27043.476} C_VEL
LIN {X 0,Y 108.092,Z 462.562,A -85,B 0,C 180,E1 -27049.443,E2 -27049.443} C_VEL
LIN {X 0,Y 101.13,Z 468.179,A -85,B 0,C 180,E1 -27056.505,E2 -27056.505} C_VEL
LIN {X 0,Y 96.215,Z 472.168,A -85,B 0,C 180,E1 -27064.005,E2 -27064.005} C_VEL
LIN {X 0,Y 92.724,Z 475.067,A -85,B 0,C 180,E1 -27072.35,E2 -27072.35} C_VEL
LIN {X 0,Y 91.061,Z 476.796,A -85,B 0,C 180,E1 -27081.119,E2 -27081.119} C_VEL
LIN {X 0,Y 90.839,Z 477.388,A -85,B 0,C 180,E1 -27089.998,E2 -27089.998} C_VEL
LIN {X 0,Y 91.06,Z 476.777,A -85,B 0,C 180,E1 -27098.878,E2 -27098.878} C_VEL
LIN {X 0,Y 92.722,Z 475.021,A -85,B 0,C 180,E1 -27107.647,E2 -27107.647} C_VEL
LIN {X 0,Y 96.218,Z 472.101,A -85,B 0,C 180,E1 -27115.99,E2 -27115.99} C_VEL
LIN {X 0,Y 101.357,Z 467.945,A -85,B 0,C 180,E1 -27123.689,E2 -27123.689} C_VEL
LIN {X 0,Y 108.086,Z 462.445,A -85,B 0,C 180,E1 -27130.555,E2 -27130.555} C_VEL
LIN {X 0,Y 116.218,Z 455.451,A -85,B 0,C 180,E1 -27136.522,E2 -27136.522} C_VEL
LIN {X 0,Y 124.132,Z 447.97,A -85,B 0,C 180,E1 -27141.119,E2 -27141.119} C_VEL
LIN {X 0,Y 132.737,Z 438.95,A -85,B 0,C 180,E1 -27145.149,E2 -27145.149} C_VEL
LIN {X 0,Y 141.77,Z 428.362,A -85,B 0,C 180,E1 -27148.562,E2 -27148.562} C_VEL
LIN {X 0,Y 142.649,Z 426.876,A -85,B 0,C 180,E1 -27149.134,E2 -27149.134} C_VEL
LIN {X 0,Y 144.573,Z 421.951,A -85,B 0,C 180,E1 -27151.641,E2 -27151.641} C_VEL
LIN {X 0,Y 145.304,Z 418.969,A -85,B 0,C 180,E1 -27153.358,E2 -27153.358} C_VEL
LIN {X 0,Y 145.859,Z 413.387,A -85,B 0,C 180,E1 -27157.328,E2 -27157.328} C_VEL
LIN {X 0,Y 146.07,Z 408.033,A -85,B 0,C 180,E1 -27161.776,E2 -27161.776} C_VEL
LIN {X 0,Y 145.978,Z 403.995,A -85,B 0,C 180,E1 -27166.071,E2 -27166.071} C_VEL
LIN {X 0,Y 145.78,Z 401.951,A -85,B 0,C 180,E1 -27168.882,E2 -27168.882} C_VEL
LIN {X 0,Y 145.533,Z 400.477,A -85,B 0,C 180,E1 -27171.67,E2 -27171.67} C_VEL
LIN {X 0,Y 145.417,Z 398.172,A -85,B 0,C 180,E1 -27180,E2 -27180} C_VEL
LIN {X 0,Y 145.371,Z 400.284,A -85,B 0,C 180,E1 -27188.34,E2 -27188.34} C_VEL
LIN {X 0,Y 145.599,Z 401.644,A -85,B 0,C 180,E1 -27191.133,E2 -27191.133} C_VEL
LIN {X 0,Y 146.092,Z 404.738,A -85,B 0,C 180,E1 -27195.826,E2 -27195.826} C_VEL
LIN {X 0,Y 146.319,Z 406.749,A -85,B 0,C 180,E1 -27198.193,E2 -27198.193} C_VEL
LIN {X 0,Y 146.329,Z 410.141,A -85,B 0,C 180,E1 -27201.295,E2 -27201.295} C_VEL
LIN {X 0,Y 145.842,Z 412.198,A -85,B 0,C 180,E1 -27202.592,E2 -27202.592} C_VEL
LIN {X 0,Y 143.607,Z 416.649,A -85,B 0,C 180,E1 -27204.353,E2 -27204.353} C_VEL
LIN {X 0,Y 140.507,Z 422.14,A -85,B 0,C 180,E1 -27206.485,E2 -27206.485} C_VEL
LIN {X 0,Y 139.866,Z 423.679,A -85,B 0,C 180,E1 -27207.354,E2 -27207.354} C_VEL
LIN {X 0,Y 138.518,Z 427.049,A -85,B 0,C 180,E1 -27209.269,E2 -27209.269} C_VEL
LIN {X 0,Y 129.299,Z 437.491,A -85,B 0,C 180,E1 -27212.599,E2 -27212.599} C_VEL
LIN {X 0,Y 120.386,Z 446.476,A -85,B 0,C 180,E1 -27216.614,E2 -27216.614} C_VEL
LIN {X 0,Y 111.887,Z 453.924,A -85,B 0,C 180,E1 -27221.086,E2 -27221.086} C_VEL
LIN {X 0,Y 103.314,Z 460.881,A -85,B 0,C 180,E1 -27227.139,E2 -27227.139} C_VEL
LIN {X 0,Y 96.002,Z 466.346,A -85,B 0,C 180,E1 -27234.153,E2 -27234.153} C_VEL
LIN {X 0,Y 90.27,Z 470.467,A -85,B 0,C 180,E1 -27242.154,E2 -27242.154} C_VEL
LIN {X 0,Y 86.275,Z 473.358,A -85,B 0,C 180,E1 -27250.986,E2 -27250.986} C_VEL
LIN {X 0,Y 84.198,Z 475.09,A -85,B 0,C 180,E1 -27260.392,E2 -27260.392} C_VEL
LIN {X 0,Y 83.813,Z 475.689,A -85,B 0,C 180,E1 -27270.002,E2 -27270.002} C_VEL
LIN {X 0,Y 84.197,Z 475.119,A -85,B 0,C 180,E1 -27279.612,E2 -27279.612} C_VEL
LIN {X 0,Y 86.242,Z 473.426,A -85,B 0,C 180,E1 -27289.026,E2 -27289.026} C_VEL
LIN {X 0,Y 90.233,Z 470.568,A -85,B 0,C 180,E1 -27297.862,E2 -27297.862} C_VEL
LIN {X 0,Y 95.946,Z 466.478,A -85,B 0,C 180,E1 -27305.875,E2 -27305.875} C_VEL
LIN {X 0,Y 103.257,Z 461.056,A -85,B 0,C 180,E1 -27312.894,E2 -27312.894} C_VEL
LIN {X 0,Y 111.821,Z 454.149,A -85,B 0,C 180,E1 -27318.957,E2 -27318.957} C_VEL
LIN {X 0,Y 120.308,Z 446.727,A -85,B 0,C 180,E1 -27323.441,E2 -27323.441} C_VEL
LIN {X 0,Y 129.221,Z 437.782,A -85,B 0,C 180,E1 -27327.459,E2 -27327.459} C_VEL
LIN {X 0,Y 138.475,Z 427.383,A -85,B 0,C 180,E1 -27330.782,E2 -27330.782} C_VEL
LIN {X 0,Y 139.846,Z 424.188,A -85,B 0,C 180,E1 -27332.55,E2 -27332.55} C_VEL
LIN {X 0,Y 140.765,Z 420.775,A -85,B 0,C 180,E1 -27334.908,E2 -27334.908} C_VEL
LIN {X 0,Y 141.38,Z 416.724,A -85,B 0,C 180,E1 -27338.11,E2 -27338.11} C_VEL
LIN {X 0,Y 141.743,Z 411.918,A -85,B 0,C 180,E1 -27342.692,E2 -27342.692} C_VEL
LIN {X 0,Y 141.644,Z 409.68,A -85,B 0,C 180,E1 -27345.635,E2 -27345.635} C_VEL
LIN {X 0,Y 141.431,Z 407.914,A -85,B 0,C 180,E1 -27348.535,E2 -27348.535} C_VEL
LIN {X 0,Y 141.293,Z 406.507,A -85,B 0,C 180,E1 -27351.418,E2 -27351.418} C_VEL
LIN {X 0,Y 141.136,Z 404.968,A -85,B 0,C 180,E1 -27357.145,E2 -27357.145} C_VEL
LIN {X 0,Y 141.445,Z 404.386,A -85,B 0,C 180,E1 -27360,E2 -27360} C_VEL
LIN {X 0,Y 141.261,Z 405.696,A -85,B 0,C 180,E1 -27365.71,E2 -27365.71} C_VEL
LIN {X 0,Y 141.461,Z 406.668,A -85,B 0,C 180,E1 -27368.571,E2 -27368.571} C_VEL
LIN {X 0,Y 141.596,Z 408.207,A -85,B 0,C 180,E1 -27371.451,E2 -27371.451} C_VEL
LIN {X 0,Y 141.544,Z 411.369,A -85,B 0,C 180,E1 -27375.519,E2 -27375.519} C_VEL
LIN {X 0,Y 141.285,Z 414.916,A -85,B 0,C 180,E1 -27379.069,E2 -27379.069} C_VEL
LIN {X 0,Y 140.558,Z 420.36,A -85,B 0,C 180,E1 -27383.578,E2 -27383.578} C_VEL
LIN {X 0,Y 139.86,Z 423.845,A -85,B 0,C 180,E1 -27386.1,E2 -27386.1} C_VEL
LIN {X 0,Y 137.74,Z 428.868,A -85,B 0,C 180,E1 -27388.881,E2 -27388.881} C_VEL
LIN {X 0,Y 135.626,Z 431.55,A -85,B 0,C 180,E1 -27389.776,E2 -27389.776} C_VEL
LIN {X 0,Y 126.151,Z 441.796,A -85,B 0,C 180,E1 -27393.314,E2 -27393.314} C_VEL
LIN {X 0,Y 118.369,Z 449.308,A -85,B 0,C 180,E1 -27396.864,E2 -27396.864} C_VEL
LIN {X 0,Y 111.442,Z 455.538,A -85,B 0,C 180,E1 -27400.819,E2 -27400.819} C_VEL
LIN {X 0,Y 102.757,Z 462.494,A -85,B 0,C 180,E1 -27406.846,E2 -27406.846} C_VEL
LIN {X 0,Y 94.783,Z 468.453,A -85,B 0,C 180,E1 -27414.649,E2 -27414.649} C_VEL
LIN {X 0,Y 89.832,Z 472.099,A -85,B 0,C 180,E1 -27422.003,E2 -27422.003} C_VEL
LIN {X 0,Y 85.923,Z 474.998,A -85,B 0,C 180,E1 -27430.901,E2 -27430.901} C_VEL
LIN {X 0,Y 84.024,Z 476.727,A -85,B 0,C 180,E1 -27440.368,E2 -27440.368} C_VEL
LIN {X 0,Y 83.76,Z 477.319,A -85,B 0,C 180,E1 -27449.998,E2 -27449.998} C_VEL
LIN {X 0,Y 84.023,Z 476.707,A -85,B 0,C 180,E1 -27459.628,E2 -27459.628} C_VEL
LIN {X 0,Y 85.922,Z 474.951,A -85,B 0,C 180,E1 -27469.096,E2 -27469.096} C_VEL
LIN {X 0,Y 89.835,Z 472.03,A -85,B 0,C 180,E1 -27477.992,E2 -27477.992} C_VEL
LIN {X 0,Y 95.472,Z 467.874,A -85,B 0,C 180,E1 -27486.077,E2 -27486.077} C_VEL
LIN {X 0,Y 102.75,Z 462.374,A -85,B 0,C 180,E1 -27493.153,E2 -27493.153} C_VEL
LIN {X 0,Y 111.438,Z 455.38,A -85,B 0,C 180,E1 -27499.18,E2 -27499.18} C_VEL
LIN {X 0,Y 119.77,Z 447.899,A -85,B 0,C 180,E1 -27503.784,E2 -27503.784} C_VEL
LIN {X 0,Y 128.794,Z 438.879,A -85,B 0,C 180,E1 -27507.754,E2 -27507.754} C_VEL
LIN {X 0,Y 136.995,Z 429.67,A -85,B 0,C 180,E1 -27510.702,E2 -27510.702} C_VEL
LIN {X 0,Y 138.17,Z 427.584,A -85,B 0,C 180,E1 -27511.713,E2 -27511.713} C_VEL
LIN {X 0,Y 139.776,Z 423.639,A -85,B 0,C 180,E1 -27513.899,E2 -27513.899} C_VEL
LIN {X 0,Y 140.62,Z 419.119,A -85,B 0,C 180,E1 -27517.212,E2 -27517.212} C_VEL
LIN {X 0,Y 141.171,Z 414.571,A -85,B 0,C 180,E1 -27521.059,E2 -27521.059} C_VEL
LIN {X 0,Y 141.38,Z 411.81,A -85,B 0,C 180,E1 -27523.768,E2 -27523.768} C_VEL
LIN {X 0,Y 141.5,Z 408.989,A -85,B 0,C 180,E1 -27527.085,E2 -27527.085} C_VEL
LIN {X 0,Y 141.492,Z 407.95,A -85,B 0,C 180,E1 -27528.54,E2 -27528.54} C_VEL
LIN {X 0,Y 141.347,Z 406.416,A -85,B 0,C 180,E1 -27531.422,E2 -27531.422} C_VEL
LIN {X 0,Y 141.061,Z 404.777,A -85,B 0,C 180,E1 -27537.145,E2 -27537.145} C_VEL
LIN {X 0,Y 141.366,Z 404.064,A -85,B 0,C 180,E1 -27540,E2 -27540} C_VEL
LIN {X 0,Y 141.089,Z 405.956,A -85,B 0,C 180,E1 -27547.743,E2 -27547.743} C_VEL
LIN {X 0,Y 141.312,Z 407.62,A -85,B 0,C 180,E1 -27551.475,E2 -27551.475} C_VEL
LIN {X 0,Y 141.567,Z 410.16,A -85,B 0,C 180,E1 -27555.447,E2 -27555.447} C_VEL
LIN {X 0,Y 141.622,Z 411.641,A -85,B 0,C 180,E1 -27557.323,E2 -27557.323} C_VEL
LIN {X 0,Y 141.454,Z 414.701,A -85,B 0,C 180,E1 -27560.352,E2 -27560.352} C_VEL
LIN {X 0,Y 140.997,Z 418.374,A -85,B 0,C 180,E1 -27563.501,E2 -27563.501} C_VEL
LIN {X 0,Y 140.127,Z 422.867,A -85,B 0,C 180,E1 -27566.833,E2 -27566.833} C_VEL
LIN {X 0,Y 139.866,Z 423.679,A -85,B 0,C 180,E1 -27567.354,E2 -27567.354} C_VEL
LIN {X 0,Y 139.011,Z 425.266,A -85,B 0,C 180,E1 -27568.073,E2 -27568.073} C_VEL
LIN {X 0,Y 136.69,Z 427.967,A -85,B 0,C 180,E1 -27568.707,E2 -27568.707} C_VEL
LIN {X 0,Y 133.788,Z 430.603,A -85,B 0,C 180,E1 -27568.985,E2 -27568.985} C_VEL
LIN {X 0,Y 128.226,Z 435.232,A -85,B 0,C 180,E1 -27569.321,E2 -27569.321} C_VEL
LIN {X 0,Y 125.239,Z 437.914,A -85,B 0,C 180,E1 -27569.989,E2 -27569.989} C_VEL
LIN {X 0,Y 116.271,Z 446.547,A -85,B 0,C 180,E1 -27573.79,E2 -27573.79} C_VEL
LIN {X 0,Y 107.325,Z 453.995,A -85,B 0,C 180,E1 -27578.209,E2 -27578.209} C_VEL
LIN {X 0,Y 98.202,Z 460.952,A -85,B 0,C 180,E1 -27584.305,E2 -27584.305} C_VEL
LIN {X 0,Y 90.282,Z 466.417,A -85,B 0,C 180,E1 -27591.485,E2 -27591.485} C_VEL
LIN {X 0,Y 84.014,Z 470.538,A -85,B 0,C 180,E1 -27599.876,E2 -27599.876} C_VEL
LIN {X 0,Y 79.567,Z 473.428,A -85,B 0,C 180,E1 -27609.312,E2 -27609.312} C_VEL
LIN {X 0,Y 77.201,Z 475.16,A -85,B 0,C 180,E1 -27619.512,E2 -27619.512} C_VEL
LIN {X 0,Y 76.734,Z 475.758,A -85,B 0,C 180,E1 -27630.002,E2 -27630.002} C_VEL
LIN {X 0,Y 77.199,Z 475.188,A -85,B 0,C 180,E1 -27640.492,E2 -27640.492} C_VEL
LIN {X 0,Y 79.537,Z 473.495,A -85,B 0,C 180,E1 -27650.7,E2 -27650.7} C_VEL
LIN {X 0,Y 83.976,Z 470.637,A -85,B 0,C 180,E1 -27660.144,E2 -27660.144} C_VEL
LIN {X 0,Y 90.245,Z 466.547,A -85,B 0,C 180,E1 -27668.538,E2 -27668.538} C_VEL
LIN {X 0,Y 98.139,Z 461.125,A -85,B 0,C 180,E1 -27675.737,E2 -27675.737} C_VEL
LIN {X 0,Y 107.263,Z 454.217,A -85,B 0,C 180,E1 -27681.838,E2 -27681.838} C_VEL
LIN {X 0,Y 116.184,Z 446.795,A -85,B 0,C 180,E1 -27686.279,E2 -27686.279} C_VEL
LIN {X 0,Y 124.145,Z 439.2,A -85,B 0,C 180,E1 -27689.692,E2 -27689.692} C_VEL
LIN {X 0,Y 132.569,Z 430.349,A -85,B 0,C 180,E1 -27692.621,E2 -27692.621} C_VEL
LIN {X 0,Y 133.914,Z 428.727,A -85,B 0,C 180,E1 -27693.149,E2 -27693.149} C_VEL
LIN {X 0,Y 134.728,Z 427.026,A -85,B 0,C 180,E1 -27694.233,E2 -27694.233} C_VEL
LIN {X 0,Y 135.781,Z 423.25,A -85,B 0,C 180,E1 -27697.159,E2 -27697.159} C_VEL
LIN {X 0,Y 136.541,Z 419.328,A -85,B 0,C 180,E1 -27700.749,E2 -27700.749} C_VEL
LIN {X 0,Y 136.925,Z 416.667,A -85,B 0,C 180,E1 -27703.602,E2 -27703.602} C_VEL
LIN {X 0,Y 136.866,Z 413.724,A -85,B 0,C 180,E1 -27708.147,E2 -27708.147} C_VEL
LIN {X 0,Y 136.838,Z 412.26,A -85,B 0,C 180,E1 -27711.136,E2 -27711.136} C_VEL
LIN {X 0,Y 136.774,Z 411.296,A -85,B 0,C 180,E1 -27714.101,E2 -27714.101} C_VEL
LIN {X 0,Y 137.156,Z 410.078,A -85,B 0,C 180,E1 -27720,E2 -27720} C_VEL
LIN {X 0,Y 136.904,Z 411.397,A -85,B 0,C 180,E1 -27725.893,E2 -27725.893} C_VEL
LIN {X 0,Y 136.992,Z 412.461,A -85,B 0,C 180,E1 -27728.853,E2 -27728.853} C_VEL
LIN {X 0,Y 136.927,Z 414.769,A -85,B 0,C 180,E1 -27732.784,E2 -27732.784} C_VEL
LIN {X 0,Y 136.601,Z 417.759,A -85,B 0,C 180,E1 -27736.437,E2 -27736.437} C_VEL
LIN {X 0,Y 135.667,Z 422.882,A -85,B 0,C 180,E1 -27741.261,E2 -27741.261} C_VEL
LIN {X 0,Y 134.566,Z 427.184,A -85,B 0,C 180,E1 -27744.697,E2 -27744.697} C_VEL
LIN {X 0,Y 133.268,Z 429.846,A -85,B 0,C 180,E1 -27746.297,E2 -27746.297} C_VEL
LIN {X 0,Y 132.226,Z 431.483,A -85,B 0,C 180,E1 -27747.09,E2 -27747.09} C_VEL
LIN {X 0,Y 122.359,Z 441.729,A -85,B 0,C 180,E1 -27750.506,E2 -27750.506} C_VEL
LIN {X 0,Y 112.985,Z 450.315,A -85,B 0,C 180,E1 -27754.589,E2 -27754.589} C_VEL
LIN {X 0,Y 104.459,Z 457.333,A -85,B 0,C 180,E1 -27759.31,E2 -27759.31} C_VEL
LIN {X 0,Y 95.536,Z 463.907,A -85,B 0,C 180,E1 -27765.663,E2 -27765.663} C_VEL
LIN {X 0,Y 88.615,Z 468.665,A -85,B 0,C 180,E1 -27772.475,E2 -27772.475} C_VEL
LIN {X 0,Y 83.565,Z 472.03,A -85,B 0,C 180,E1 -27779.693,E2 -27779.693} C_VEL
LIN {X 0,Y 79.19,Z 474.928,A -85,B 0,C 180,E1 -27789.205,E2 -27789.205} C_VEL
LIN {X 0,Y 76.994,Z 476.658,A -85,B 0,C 180,E1 -27799.479,E2 -27799.479} C_VEL
LIN {X 0,Y 76.671,Z 477.25,A -85,B 0,C 180,E1 -27809.998,E2 -27809.998} C_VEL
LIN {X 0,Y 76.993,Z 476.638,A -85,B 0,C 180,E1 -27820.517,E2 -27820.517} C_VEL
LIN {X 0,Y 79.189,Z 474.881,A -85,B 0,C 180,E1 -27830.791,E2 -27830.791} C_VEL
LIN {X 0,Y 83.569,Z 471.96,A -85,B 0,C 180,E1 -27840.301,E2 -27840.301} C_VEL
LIN {X 0,Y 89.795,Z 467.804,A -85,B 0,C 180,E1 -27848.762,E2 -27848.762} C_VEL
LIN {X 0,Y 97.653,Z 462.303,A -85,B 0,C 180,E1 -27856.026,E2 -27856.026} C_VEL
LIN {X 0,Y 106.902,Z 455.309,A -85,B 0,C 180,E1 -27862.08,E2 -27862.08} C_VEL
LIN {X 0,Y 116.002,Z 447.54,A -85,B 0,C 180,E1 -27866.79,E2 -27866.79} C_VEL
LIN {X 0,Y 125.124,Z 438.807,A -85,B 0,C 180,E1 -27870.525,E2 -27870.525} C_VEL
LIN {X 0,Y 132.197,Z 431.228,A -85,B 0,C 180,E1 -27872.929,E2 -27872.929} C_VEL
LIN {X 0,Y 134.08,Z 427.942,A -85,B 0,C 180,E1 -27874.706,E2 -27874.706} C_VEL
LIN {X 0,Y 134.825,Z 425.787,A -85,B 0,C 180,E1 -27876.173,E2 -27876.173} C_VEL
LIN {X 0,Y 135.915,Z 420.902,A -85,B 0,C 180,E1 -27880.297,E2 -27880.297} C_VEL
LIN {X 0,Y 136.498,Z 417.552,A -85,B 0,C 180,E1 -27883.55,E2 -27883.55} C_VEL
LIN {X 0,Y 136.886,Z 413.853,A -85,B 0,C 180,E1 -27888.149,E2 -27888.149} C_VEL
LIN {X 0,Y 136.892,Z 412.213,A -85,B 0,C 180,E1 -27891.14,E2 -27891.14} C_VEL
LIN {X 0,Y 136.801,Z 411.145,A -85,B 0,C 180,E1 -27894.103,E2 -27894.103} C_VEL
LIN {X 0,Y 137.085,Z 409.768,A -85,B 0,C 180,E1 -27900,E2 -27900} C_VEL
LIN {X 0,Y 136.67,Z 411.02,A -85,B 0,C 180,E1 -27905.903,E2 -27905.903} C_VEL
LIN {X 0,Y 136.726,Z 411.987,A -85,B 0,C 180,E1 -27908.871,E2 -27908.871} C_VEL
LIN {X 0,Y 136.771,Z 413.802,A -85,B 0,C 180,E1 -27912.504,E2 -27912.504} C_VEL
LIN {X 0,Y 136.814,Z 416.402,A -85,B 0,C 180,E1 -27916.412,E2 -27916.412} C_VEL
LIN {X 0,Y 136.312,Z 419.901,A -85,B 0,C 180,E1 -27920.098,E2 -27920.098} C_VEL
LIN {X 0,Y 135.158,Z 425.098,A -85,B 0,C 180,E1 -27924.582,E2 -27924.582} C_VEL
LIN {X 0,Y 133.918,Z 428.384,A -85,B 0,C 180,E1 -27926.859,E2 -27926.859} C_VEL
LIN {X 0,Y 131.218,Z 431.629,A -85,B 0,C 180,E1 -27927.908,E2 -27927.908} C_VEL
LIN {X 0,Y 125.239,Z 437.914,A -85,B 0,C 180,E1 -27929.989,E2 -27929.989} C_VEL
LIN {X 0,Y 121.224,Z 441.558,A -85,B 0,C 180,E1 -27931.156,E2 -27931.156} C_VEL
LIN {X 0,Y 113.524,Z 447.176,A -85,B 0,C 180,E1 -27932.536,E2 -27932.536} C_VEL
LIN {X 0,Y 105.693,Z 452.321,A -85,B 0,C 180,E1 -27934.214,E2 -27934.214} C_VEL
LIN {X 0,Y 101.566,Z 455.175,A -85,B 0,C 180,E1 -27935.921,E2 -27935.921} C_VEL
LIN {X 0,Y 93.35,Z 461.023,A -85,B 0,C 180,E1 -27941.165,E2 -27941.165} C_VEL
LIN {X 0,Y 84.772,Z 466.488,A -85,B 0,C 180,E1 -27948.456,E2 -27948.456} C_VEL
LIN {X 0,Y 77.916,Z 470.608,A -85,B 0,C 180,E1 -27957.238,E2 -27957.238} C_VEL
LIN {X 0,Y 72.927,Z 473.498,A -85,B 0,C 180,E1 -27967.329,E2 -27967.329} C_VEL
LIN {X 0,Y 70.211,Z 475.229,A -85,B 0,C 180,E1 -27978.454,E2 -27978.454} C_VEL
LIN {X 0,Y 69.646,Z 475.827,A -85,B 0,C 180,E1 -27990.002,E2 -27990.002} C_VEL
LIN {X 0,Y 70.208,Z 475.257,A -85,B 0,C 180,E1 -28001.551,E2 -28001.551} C_VEL
LIN {X 0,Y 72.898,Z 473.564,A -85,B 0,C 180,E1 -28012.685,E2 -28012.685} C_VEL
LIN {X 0,Y 77.878,Z 470.705,A -85,B 0,C 180,E1 -28022.785,E2 -28022.785} C_VEL
LIN {X 0,Y 85.317,Z 466.254,A -85,B 0,C 180,E1 -28032.15,E2 -28032.15} C_VEL
LIN {X 0,Y 93.296,Z 461.193,A -85,B 0,C 180,E1 -28038.878,E2 -28038.878} C_VEL
LIN {X 0,Y 103.005,Z 454.285,A -85,B 0,C 180,E1 -28044.961,E2 -28044.961} C_VEL
LIN {X 0,Y 112.368,Z 446.863,A -85,B 0,C 180,E1 -28049.316,E2 -28049.316} C_VEL
LIN {X 0,Y 122.13,Z 437.917,A -85,B 0,C 180,E1 -28053.121,E2 -28053.121} C_VEL
LIN {X 0,Y 127.966,Z 432.036,A -85,B 0,C 180,E1 -28054.985,E2 -28054.985} C_VEL
LIN {X 0,Y 129.277,Z 430.42,A -85,B 0,C 180,E1 -28055.589,E2 -28055.589} C_VEL
LIN {X 0,Y 130.348,Z 427.692,A -85,B 0,C 180,E1 -28057.826,E2 -28057.826} C_VEL
LIN {X 0,Y 131.327,Z 424.121,A -85,B 0,C 180,E1 -28061.271,E2 -28061.271} C_VEL
LIN {X 0,Y 131.972,Z 421.3,A -85,B 0,C 180,E1 -28064.557,E2 -28064.557} C_VEL
LIN {X 0,Y 132.072,Z 419.33,A -85,B 0,C 180,E1 -28067.71,E2 -28067.71} C_VEL
LIN {X 0,Y 132.12,Z 417.861,A -85,B 0,C 180,E1 -28070.817,E2 -28070.817} C_VEL
LIN {X 0,Y 132.165,Z 416.828,A -85,B 0,C 180,E1 -28073.895,E2 -28073.895} C_VEL
LIN {X 0,Y 132.624,Z 415.593,A -85,B 0,C 180,E1 -28080,E2 -28080} C_VEL
LIN {X 0,Y 132.295,Z 416.944,A -85,B 0,C 180,E1 -28086.099,E2 -28086.099} C_VEL
LIN {X 0,Y 132.257,Z 418.098,A -85,B 0,C 180,E1 -28089.173,E2 -28089.173} C_VEL
LIN {X 0,Y 131.931,Z 420.584,A -85,B 0,C 180,E1 -28093.277,E2 -28093.277} C_VEL
LIN {X 0,Y 131.527,Z 422.687,A -85,B 0,C 180,E1 -28095.885,E2 -28095.885} C_VEL
LIN {X 0,Y 130.484,Z 426.63,A -85,B 0,C 180,E1 -28099.897,E2 -28099.897} C_VEL
LIN {X 0,Y 129.492,Z 429.76,A -85,B 0,C 180,E1 -28102.683,E2 -28102.683} C_VEL
LIN {X 0,Y 128.901,Z 431.102,A -85,B 0,C 180,E1 -28103.682,E2 -28103.682} C_VEL
LIN {X 0,Y 127.643,Z 433.043,A -85,B 0,C 180,E1 -28104.702,E2 -28104.702} C_VEL
LIN {X 0,Y 117.469,Z 443.015,A -85,B 0,C 180,E1 -28108.057,E2 -28108.057} C_VEL
LIN {X 0,Y 109.475,Z 449.913,A -85,B 0,C 180,E1 -28111.302,E2 -28111.302} C_VEL
LIN {X 0,Y 102.66,Z 455.402,A -85,B 0,C 180,E1 -28114.763,E2 -28114.763} C_VEL
LIN {X 0,Y 92.835,Z 462.357,A -85,B 0,C 180,E1 -28120.794,E2 -28120.794} C_VEL
LIN {X 0,Y 84.282,Z 467.825,A -85,B 0,C 180,E1 -28128.155,E2 -28128.155} C_VEL
LIN {X 0,Y 77.456,Z 471.961,A -85,B 0,C 180,E1 -28137.014,E2 -28137.014} C_VEL
LIN {X 0,Y 72.541,Z 474.859,A -85,B 0,C 180,E1 -28147.197,E2 -28147.197} C_VEL
LIN {X 0,Y 70.001,Z 476.589,A -85,B 0,C 180,E1 -28158.414,E2 -28158.414} C_VEL
LIN {X 0,Y 69.571,Z 477.181,A -85,B 0,C 180,E1 -28169.998,E2 -28169.998} C_VEL
LIN {X 0,Y 69.999,Z 476.568,A -85,B 0,C 180,E1 -28181.581,E2 -28181.581} C_VEL
LIN {X 0,Y 72.54,Z 474.811,A -85,B 0,C 180,E1 -28192.799,E2 -28192.799} C_VEL
LIN {X 0,Y 77.462,Z 471.89,A -85,B 0,C 180,E1 -28202.979,E2 -28202.979} C_VEL
LIN {X 0,Y 84.325,Z 467.733,A -85,B 0,C 180,E1 -28211.814,E2 -28211.814} C_VEL
LIN {X 0,Y 92.81,Z 462.232,A -85,B 0,C 180,E1 -28219.218,E2 -28219.218} C_VEL
LIN {X 0,Y 102.653,Z 455.238,A -85,B 0,C 180,E1 -28225.238,E2 -28225.238} C_VEL
LIN {X 0,Y 111.589,Z 448.02,A -85,B 0,C 180,E1 -28229.576,E2 -28229.576} C_VEL
LIN {X 0,Y 121.763,Z 438.735,A -85,B 0,C 180,E1 -28233.458,E2 -28233.458} C_VEL
LIN {X 0,Y 127.624,Z 432.786,A -85,B 0,C 180,E1 -28235.311,E2 -28235.311} C_VEL
LIN {X 0,Y 129.169,Z 430.225,A -85,B 0,C 180,E1 -28236.769,E2 -28236.769} C_VEL
LIN {X 0,Y 130.411,Z 426.372,A -85,B 0,C 180,E1 -28240.141,E2 -28240.141} C_VEL
LIN {X 0,Y 131.53,Z 422.123,A -85,B 0,C 180,E1 -28244.505,E2 -28244.505} C_VEL
LIN {X 0,Y 131.963,Z 419.639,A -85,B 0,C 180,E1 -28247.7,E2 -28247.7} C_VEL
LIN {X 0,Y 132.163,Z 417.862,A -85,B 0,C 180,E1 -28250.821,E2 -28250.821} C_VEL
LIN {X 0,Y 132.215,Z 416.687,A -85,B 0,C 180,E1 -28253.898,E2 -28253.898} C_VEL
LIN {X 0,Y 132.556,Z 415.285,A -85,B 0,C 180,E1 -28260,E2 -28260} C_VEL
LIN {X 0,Y 132.071,Z 416.562,A -85,B 0,C 180,E1 -28266.11,E2 -28266.11} C_VEL
LIN {X 0,Y 132.03,Z 417.584,A -85,B 0,C 180,E1 -28269.189,E2 -28269.189} C_VEL
LIN {X 0,Y 131.956,Z 419.077,A -85,B 0,C 180,E1 -28272.301,E2 -28272.301} C_VEL
LIN {X 0,Y 131.744,Z 421.653,A -85,B 0,C 180,E1 -28276.222,E2 -28276.222} C_VEL
LIN {X 0,Y 130.804,Z 425.55,A -85,B 0,C 180,E1 -28280.441,E2 -28280.441} C_VEL
LIN {X 0,Y 129.573,Z 429.288,A -85,B 0,C 180,E1 -28283.766,E2 -28283.766} C_VEL
LIN {X 0,Y 129.046,Z 430.488,A -85,B 0,C 180,E1 -28284.666,E2 -28284.666} C_VEL
LIN {X 0,Y 122.195,Z 437.635,A -85,B 0,C 180,E1 -28286.945,E2 -28286.945} C_VEL
LIN {X 0,Y 112.448,Z 446.618,A -85,B 0,C 180,E1 -28290.757,E2 -28290.757} C_VEL
LIN {X 0,Y 103.059,Z 454.066,A -85,B 0,C 180,E1 -28295.086,E2 -28295.086} C_VEL
LIN {X 0,Y 101.566,Z 455.175,A -85,B 0,C 180,E1 -28295.921,E2 -28295.921} C_VEL
